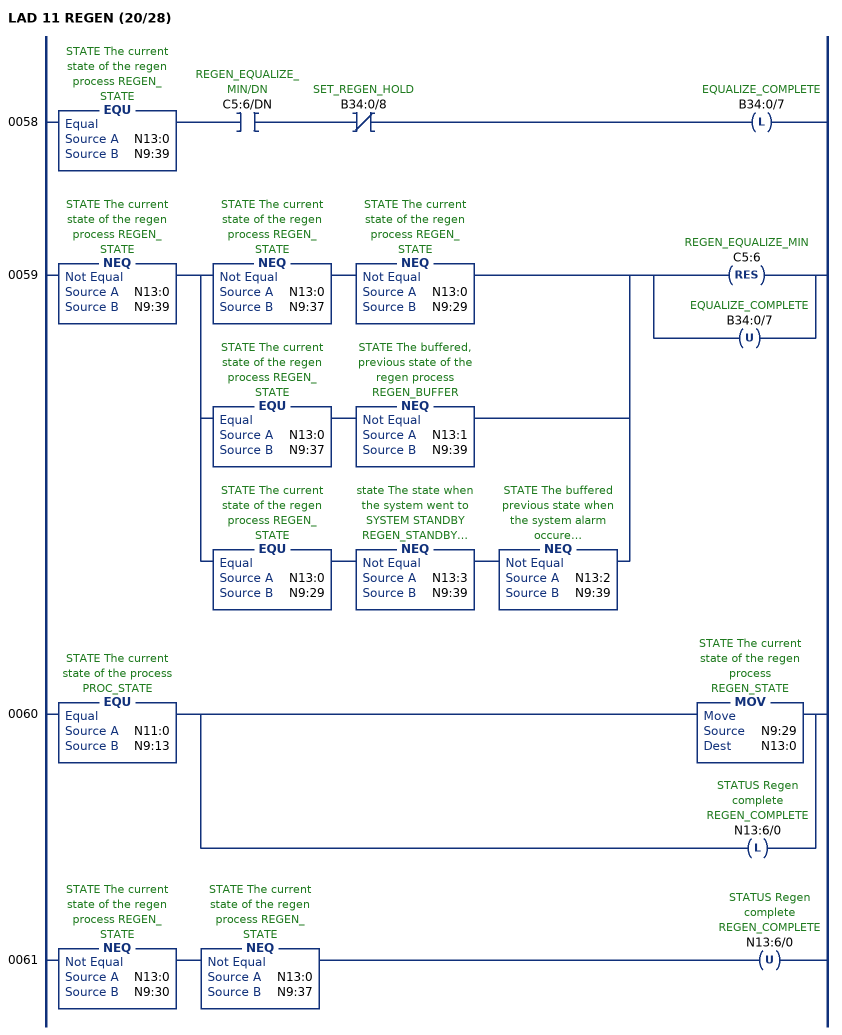
% Rung: 58 %
SOR EQU N13:0 N9:39 XIC C5:6/DN XIO B34:0/8 OTL B34:0/7 EOR
%   N13:0  REGEN_STATE  "STATE The current state of the regen process" %
%   N9:39  REGEN_EQUALIZE %
%   C5:6  REGEN_EQUALIZE_MIN %
%   B34:0/8  SET_REGEN_HOLD %
%   B34:0/7  EQUALIZE_COMPLETE %
% Rung: 59 %
SOR NEQ N13:0 N9:39 BST NEQ N13:0 N9:37 NEQ N13:0 N9:29 NXB EQU N13:0 N9:37 NEQ N13:1 N9:39 NXB EQU N13:0 N9:29 NEQ N13:3 N9:39 NEQ N13:2 N9:39 BND BST RES C5:6 NXB OTU B34:0/7 BND EOR
%   N13:0  REGEN_STATE  "STATE The current state of the regen process" %
%   N9:39  REGEN_EQUALIZE %
%   N9:37  REGEN_ALARM  "STATE Regen Alarm" %
%   N9:29  REGEN_IDLE %
%   N13:1  REGEN_BUFFER  "STATE The buffered, previous state of the regen process" %
%   N13:3  REGEN_STANDBY_BUFFER  "state The state when the system went to SYSTEM STANDBY" %
%   N13:2  REGEN_ALARM_BUFFER  "STATE The buffered previous state when the system alarm occured" %
%   C5:6  REGEN_EQUALIZE_MIN %
%   B34:0/7  EQUALIZE_COMPLETE %
% Rung: 60 %
SOR EQU N11:0 N9:13 BST MOV N9:29 N13:0 NXB OTL N13:6/0 BND EOR
%   N11:0  PROC_STATE  "STATE The current state of the process" %
%   N9:13  PROC_OVERLAP  "STATE Process Purify Overlap" %
%   N9:29  REGEN_IDLE %
%   N13:0  REGEN_STATE  "STATE The current state of the regen process" %
%   N13:6/0  REGEN_COMPLETE  "STATUS Regen complete" %
% Rung: 61 %
SOR NEQ N13:0 N9:30 NEQ N13:0 N9:37 OTU N13:6/0 EOR
%   N13:0  REGEN_STATE  "STATE The current state of the regen process" %
%   N9:30  REGEN_STANDBY  "STATE Regen Standby" %
%   N9:37  REGEN_ALARM  "STATE Regen Alarm" %
%   N13:6/0  REGEN_COMPLETE  "STATUS Regen complete" %

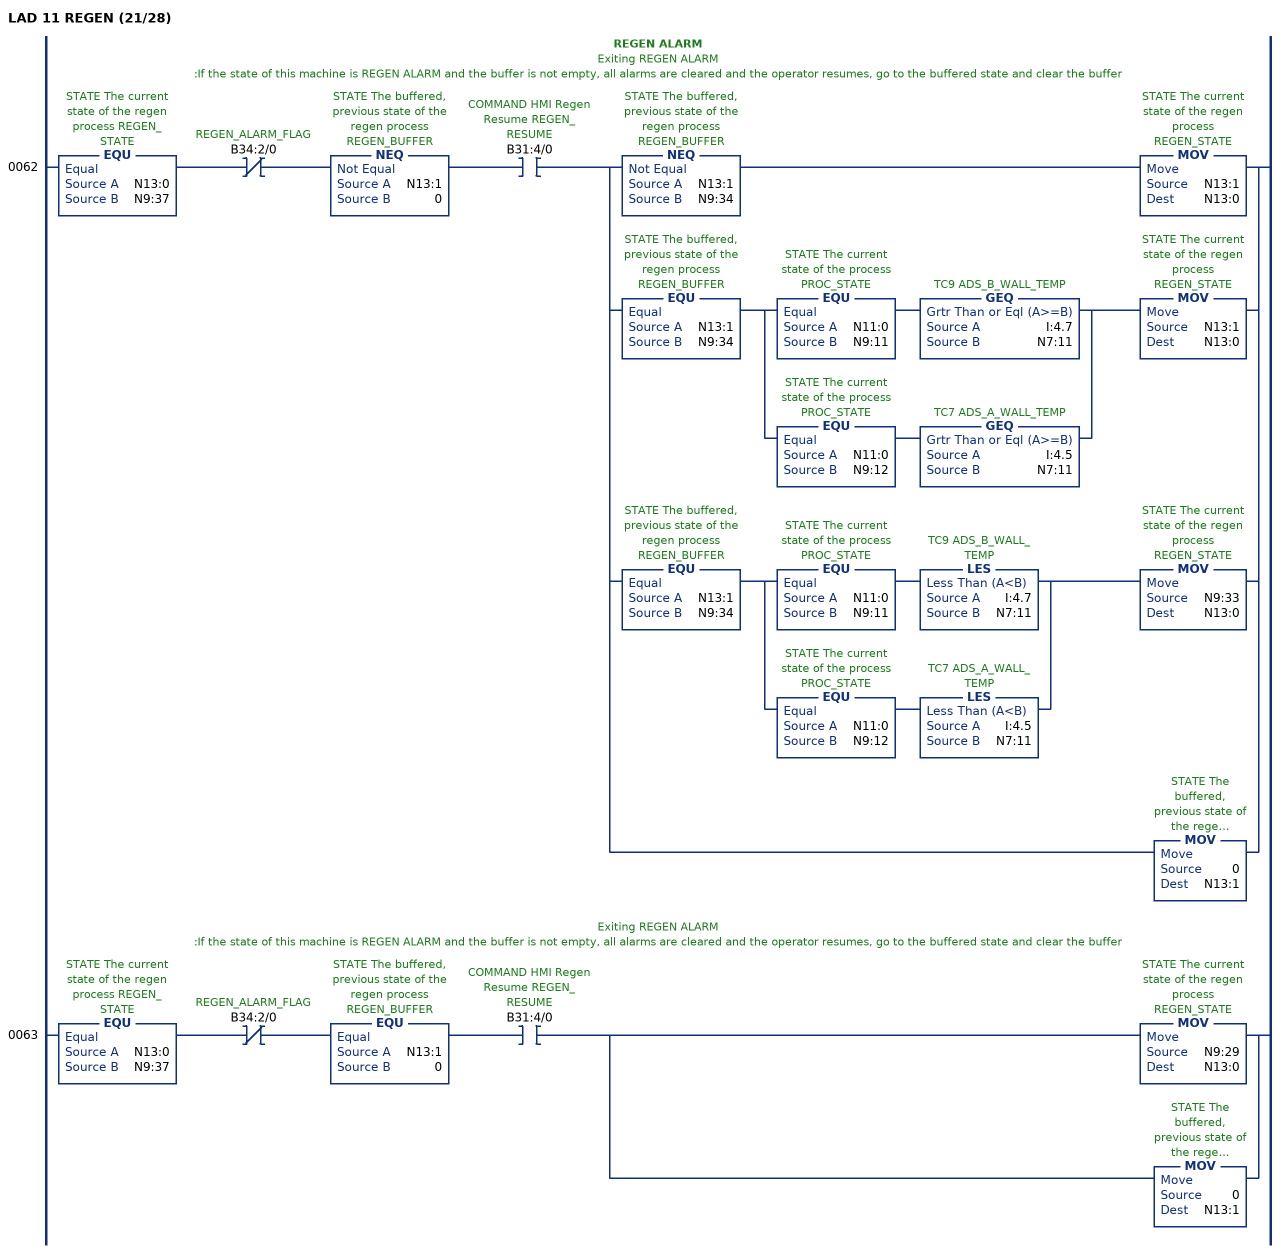
% Rung: 62 %
% TITLE: REGEN ALARM %
% Exiting REGEN ALARM
% :If the state of this machine is REGEN ALARM and the buffer is not empty, all alarms are cleared and the operator resumes, go to the buffered state and clear the buffer %
SOR EQU N13:0 N9:37 XIO B34:2/0 NEQ N13:1 0 XIC B31:4/0 BST NEQ N13:1 N9:34 MOV N13:1 N13:0 NXB EQU N13:1 N9:34 BST EQU N11:0 N9:11 GEQ I:4.7 N7:11 NXB EQU N11:0 N9:12 GEQ I:4.5 N7:11 BND MOV N13:1 N13:0 NXB EQU N13:1 N9:34 BST EQU N11:0 N9:11 LES I:4.7 N7:11 NXB EQU N11:0 N9:12 LES I:4.5 N7:11 BND MOV N9:33 N13:0 NXB MOV 0 N13:1 BND EOR
%   N13:0  REGEN_STATE  "STATE The current state of the regen process" %
%   N9:37  REGEN_ALARM  "STATE Regen Alarm" %
%   B34:2/0  REGEN_ALARM_FLAG %
%   N13:1  REGEN_BUFFER  "STATE The buffered, previous state of the regen process" %
%   B31:4/0  REGEN_RESUME  "COMMAND HMI Regen Resume" %
%   N9:34  REGEN_H2_REDUCTION  "STATE Regen Running" %
%   N11:0  PROC_STATE  "STATE The current state of the process" %
%   N9:11  PROC_PURIFY_A  "STATE Process Purify A" %
%   I:4.7  ADS_B_WALL_TEMP  "TC9" %
%   N7:11  ADS_BED_TEMP_HIGH  "CONFIG The temp at which the regen process may continue" %
%   N9:12  PROC_PURIFY_B  "STATE Process Purify B" %
%   I:4.5  ADS_A_WALL_TEMP  "TC7" %
%   N9:33  REGEN_HEAT_BED  "STATE Regen Heat wall" %
% Rung: 63 %
% Exiting REGEN ALARM
% :If the state of this machine is REGEN ALARM and the buffer is not empty, all alarms are cleared and the operator resumes, go to the buffered state and clear the buffer %
SOR EQU N13:0 N9:37 XIO B34:2/0 EQU N13:1 0 XIC B31:4/0 BST MOV N9:29 N13:0 NXB MOV 0 N13:1 BND EOR
%   N13:0  REGEN_STATE  "STATE The current state of the regen process" %
%   N9:37  REGEN_ALARM  "STATE Regen Alarm" %
%   B34:2/0  REGEN_ALARM_FLAG %
%   N13:1  REGEN_BUFFER  "STATE The buffered, previous state of the regen process" %
%   B31:4/0  REGEN_RESUME  "COMMAND HMI Regen Resume" %
%   N9:29  REGEN_IDLE %

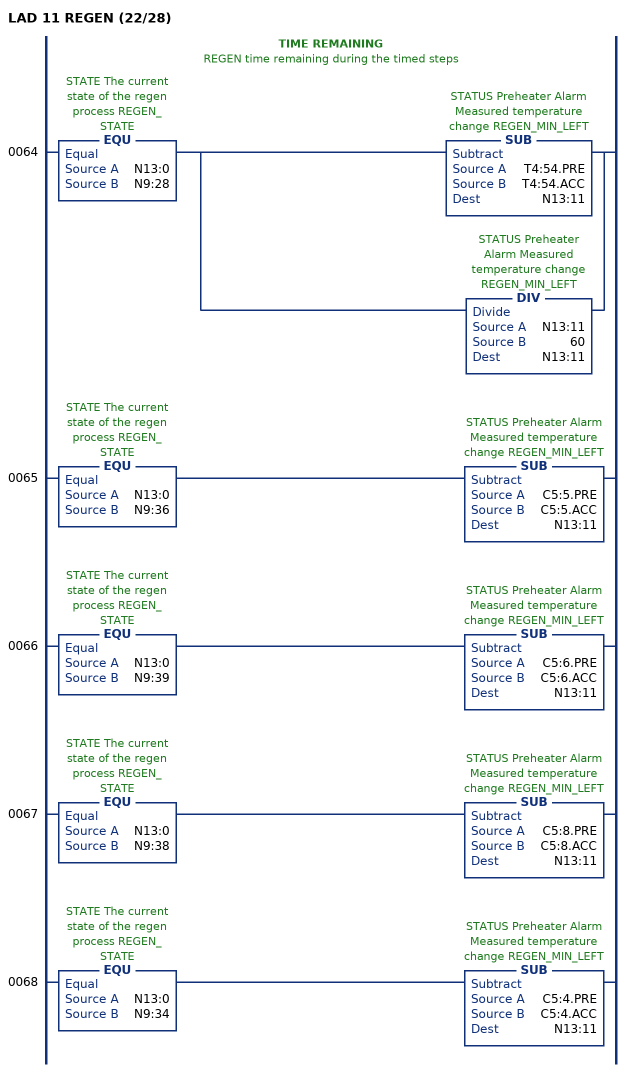
% Rung: 64 %
% TITLE: TIME REMAINING %
% REGEN time remaining during the timed steps %
SOR EQU N13:0 N9:28 BST SUB T4:54.PRE T4:54.ACC N13:11 NXB DIV N13:11 60 N13:11 BND EOR
%   N13:0  REGEN_STATE  "STATE The current state of the regen process" %
%   N9:28  REGEN_VENT_2  "STATE Regen Vent 2" %
%   T4:54  REGEN_VENT_2_TMR %
%   N13:11  REGEN_MIN_LEFT  "STATUS Preheater Alarm Measured temperature change" %
% Rung: 65 %
SOR EQU N13:0 N9:36 SUB C5:5.PRE C5:5.ACC N13:11 EOR
%   N13:0  REGEN_STATE  "STATE The current state of the regen process" %
%   N9:36  REGEN_COOL  "STATE Regen Cool" %
%   C5:5  REGEN_COOL_MINUTE  "COUNTER Regen the number of minutes for which the bed has cooled" %
%   N13:11  REGEN_MIN_LEFT  "STATUS Preheater Alarm Measured temperature change" %
% Rung: 66 %
SOR EQU N13:0 N9:39 SUB C5:6.PRE C5:6.ACC N13:11 EOR
%   N13:0  REGEN_STATE  "STATE The current state of the regen process" %
%   N9:39  REGEN_EQUALIZE %
%   C5:6  REGEN_EQUALIZE_MIN %
%   N13:11  REGEN_MIN_LEFT  "STATUS Preheater Alarm Measured temperature change" %
% Rung: 67 %
SOR EQU N13:0 N9:38 SUB C5:8.PRE C5:8.ACC N13:11 EOR
%   N13:0  REGEN_STATE  "STATE The current state of the regen process" %
%   N9:38  REGEN_PURGE  "STATE Regen Hot Purge" %
%   C5:8  REGEN_PURGE_MINUTES  "COUNTER Regen THe number of minutes the purge step runs" %
%   N13:11  REGEN_MIN_LEFT  "STATUS Preheater Alarm Measured temperature change" %
% Rung: 68 %
SOR EQU N13:0 N9:34 SUB C5:4.PRE C5:4.ACC N13:11 EOR
%   N13:0  REGEN_STATE  "STATE The current state of the regen process" %
%   N9:34  REGEN_H2_REDUCTION  "STATE Regen Running" %
%   C5:4  REGEN_REDUC_MINUTE  "COUNTER Regen The number of minutes which the regen reduc runs" %
%   N13:11  REGEN_MIN_LEFT  "STATUS Preheater Alarm Measured temperature change" %

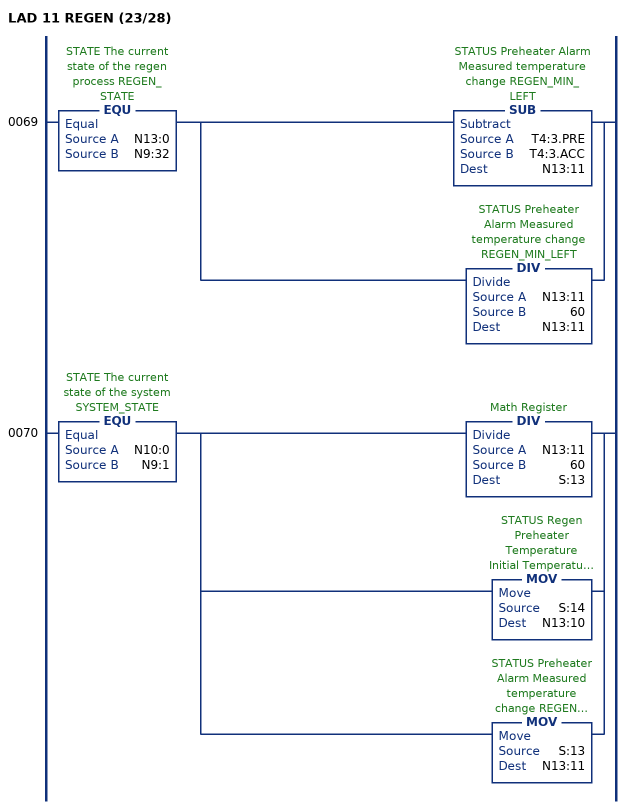
% Rung: 69 %
SOR EQU N13:0 N9:32 BST SUB T4:3.PRE T4:3.ACC N13:11 NXB DIV N13:11 60 N13:11 BND EOR
%   N13:0  REGEN_STATE  "STATE The current state of the regen process" %
%   N9:32  REGEN_VENT  "STATE Regen Vent" %
%   T4:3  REGEN_VENT_TIMER  "TIMER Regen Vent (seconds)" %
%   N13:11  REGEN_MIN_LEFT  "STATUS Preheater Alarm Measured temperature change" %
% Rung: 70 %
SOR EQU N10:0 N9:1 BST DIV N13:11 60 S:13 NXB MOV S:14 N13:10 NXB MOV S:13 N13:11 BND EOR
%   N10:0  SYSTEM_STATE  "STATE The current state of the system" %
%   N9:1  SYSTEM_PROCESS  "STATE System Process" %
%   N13:11  REGEN_MIN_LEFT  "STATUS Preheater Alarm Measured temperature change" %
%   S:13  "Math Register" %
%   S:14  "Math Register" %
%   N13:10  REGEN_HRS_LEFT  "STATUS Regen Preheater Temperature Initial Temperature" %

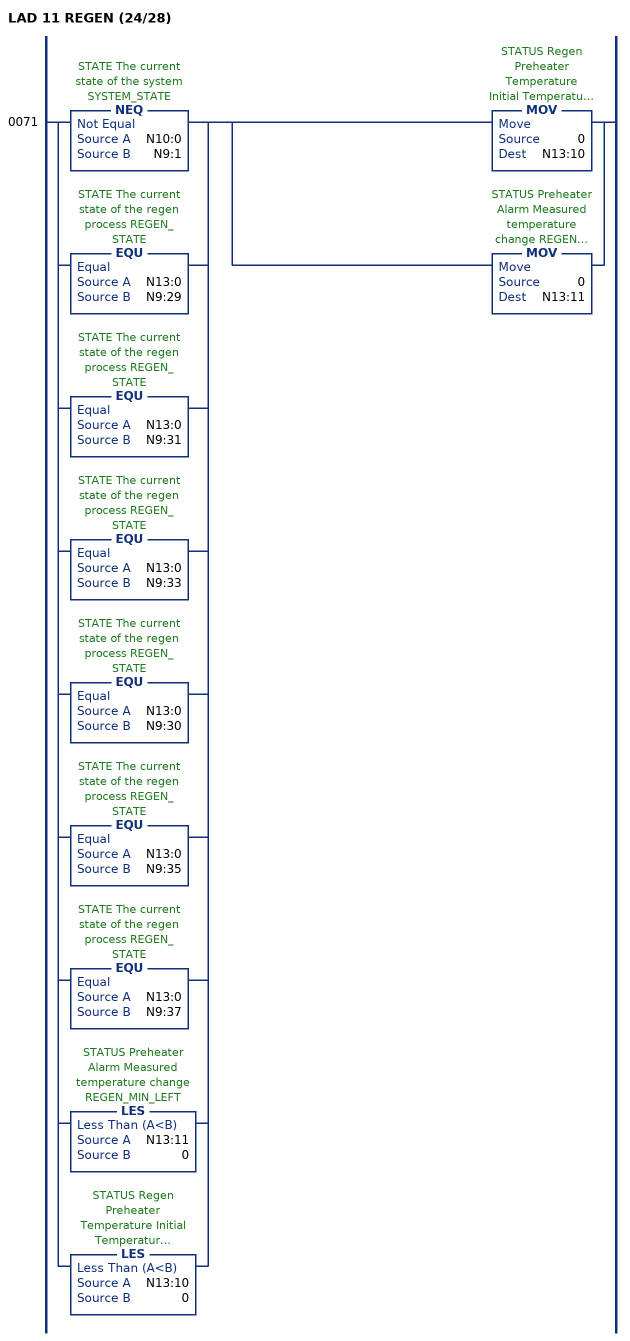
% Rung: 71 %
SOR BST NEQ N10:0 N9:1 NXB EQU N13:0 N9:29 NXB EQU N13:0 N9:31 NXB EQU N13:0 N9:33 NXB EQU N13:0 N9:30 NXB EQU N13:0 N9:35 NXB EQU N13:0 N9:37 NXB LES N13:11 0 NXB LES N13:10 0 BND BST MOV 0 N13:10 NXB MOV 0 N13:11 BND EOR
%   N10:0  SYSTEM_STATE  "STATE The current state of the system" %
%   N9:1  SYSTEM_PROCESS  "STATE System Process" %
%   N13:0  REGEN_STATE  "STATE The current state of the regen process" %
%   N9:29  REGEN_IDLE %
%   N9:31  REGEN_DELAY  "STATE Regen Delay" %
%   N9:33  REGEN_HEAT_BED  "STATE Regen Heat wall" %
%   N9:30  REGEN_STANDBY  "STATE Regen Standby" %
%   N9:35  REGEN_COOL_WALL  "STATE Regen Cool wall" %
%   N9:37  REGEN_ALARM  "STATE Regen Alarm" %
%   N13:11  REGEN_MIN_LEFT  "STATUS Preheater Alarm Measured temperature change" %
%   N13:10  REGEN_HRS_LEFT  "STATUS Regen Preheater Temperature Initial Temperature" %

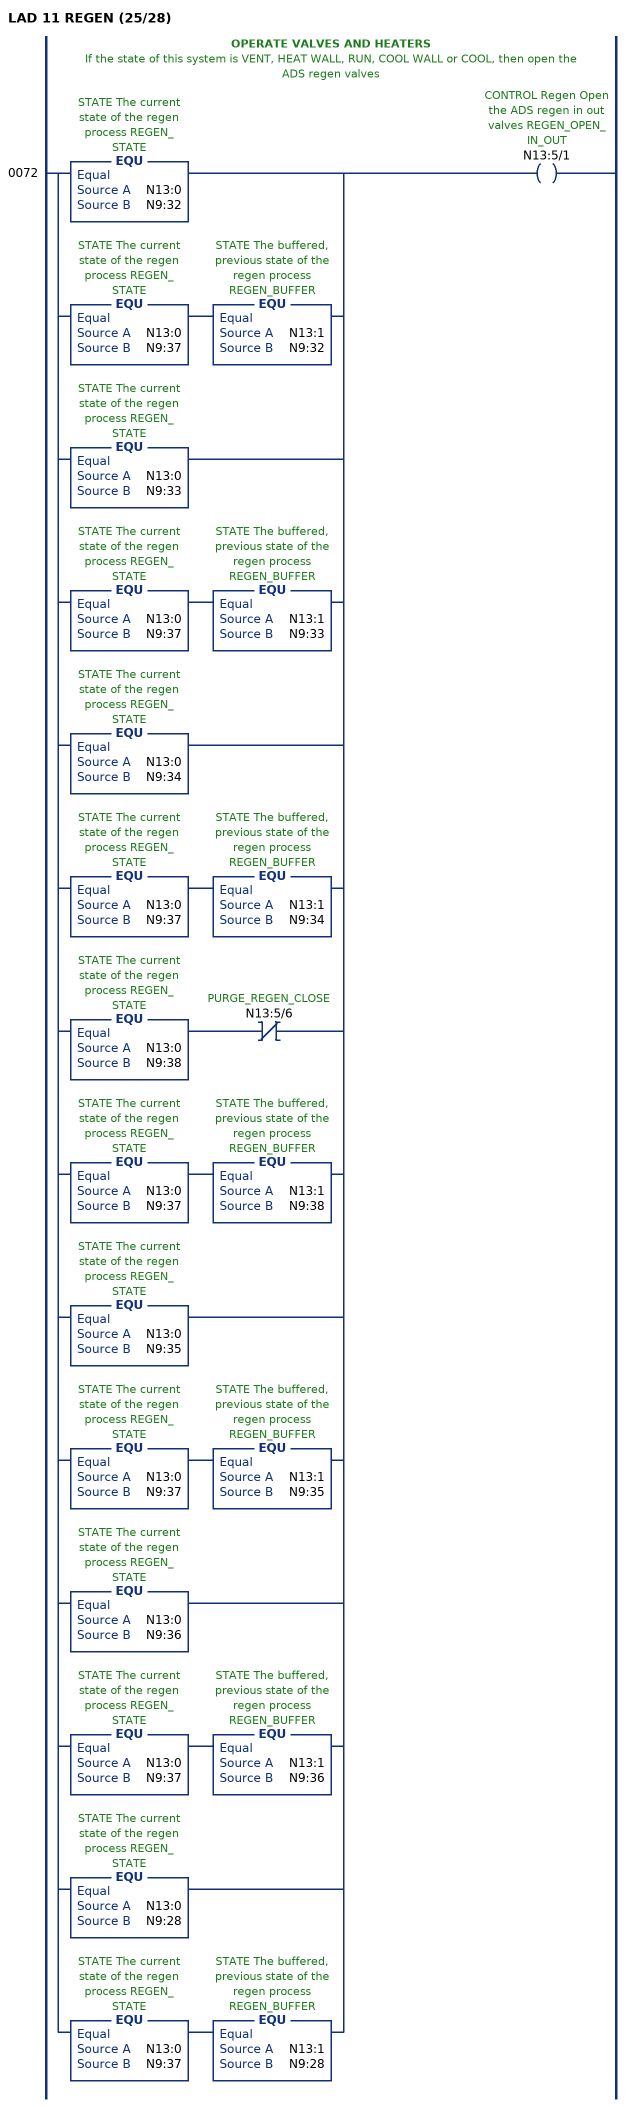
% Rung: 72 %
% TITLE: OPERATE VALVES AND HEATERS %
% If the state of this system is VENT, HEAT WALL, RUN, COOL WALL or COOL, then open the ADS regen valves %
SOR BST EQU N13:0 N9:32 NXB EQU N13:0 N9:37 EQU N13:1 N9:32 NXB EQU N13:0 N9:33 NXB EQU N13:0 N9:37 EQU N13:1 N9:33 NXB EQU N13:0 N9:34 NXB EQU N13:0 N9:37 EQU N13:1 N9:34 NXB EQU N13:0 N9:38 XIO N13:5/6 NXB EQU N13:0 N9:37 EQU N13:1 N9:38 NXB EQU N13:0 N9:35 NXB EQU N13:0 N9:37 EQU N13:1 N9:35 NXB EQU N13:0 N9:36 NXB EQU N13:0 N9:37 EQU N13:1 N9:36 NXB EQU N13:0 N9:28 NXB EQU N13:0 N9:37 EQU N13:1 N9:28 BND OTE N13:5/1 EOR
%   N13:0  REGEN_STATE  "STATE The current state of the regen process" %
%   N9:32  REGEN_VENT  "STATE Regen Vent" %
%   N9:37  REGEN_ALARM  "STATE Regen Alarm" %
%   N13:1  REGEN_BUFFER  "STATE The buffered, previous state of the regen process" %
%   N9:33  REGEN_HEAT_BED  "STATE Regen Heat wall" %
%   N9:34  REGEN_H2_REDUCTION  "STATE Regen Running" %
%   N9:38  REGEN_PURGE  "STATE Regen Hot Purge" %
%   N13:5/6  PURGE_REGEN_CLOSE %
%   N9:35  REGEN_COOL_WALL  "STATE Regen Cool wall" %
%   N9:36  REGEN_COOL  "STATE Regen Cool" %
%   N9:28  REGEN_VENT_2  "STATE Regen Vent 2" %
%   N13:5/1  REGEN_OPEN_IN_OUT  "CONTROL Regen Open the ADS regen in out valves" %

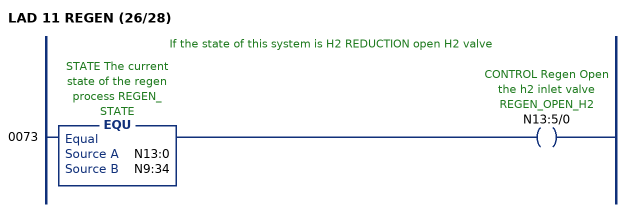
% Rung: 73 %
% If the state of this system is H2 REDUCTION open H2 valve %
SOR EQU N13:0 N9:34 OTE N13:5/0 EOR
%   N13:0  REGEN_STATE  "STATE The current state of the regen process" %
%   N9:34  REGEN_H2_REDUCTION  "STATE Regen Running" %
%   N13:5/0  REGEN_OPEN_H2  "CONTROL Regen Open the h2 inlet valve" %

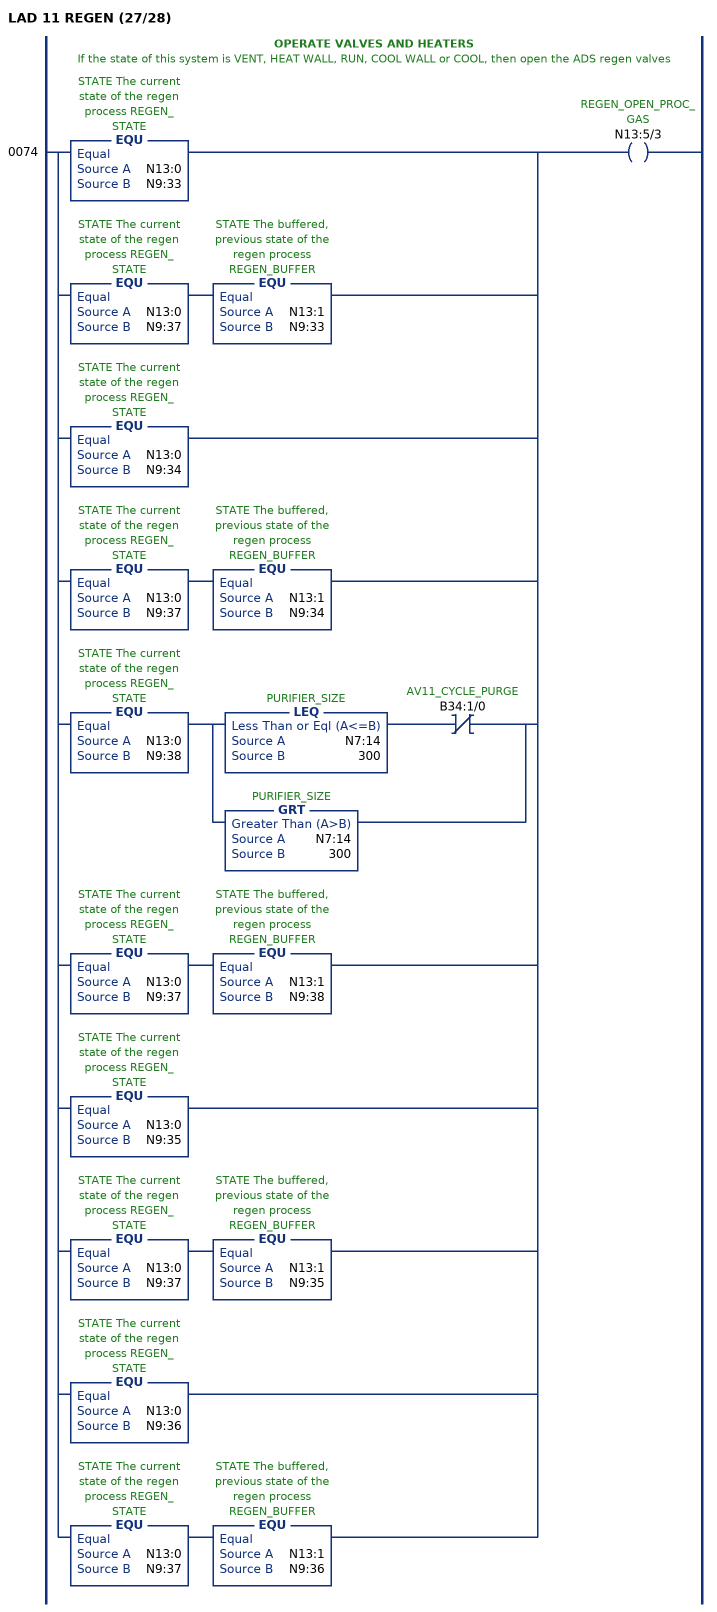
% Rung: 74 %
% TITLE: OPERATE VALVES AND HEATERS %
% If the state of this system is VENT, HEAT WALL, RUN, COOL WALL or COOL, then open the ADS regen valves %
SOR BST EQU N13:0 N9:33 NXB EQU N13:0 N9:37 EQU N13:1 N9:33 NXB EQU N13:0 N9:34 NXB EQU N13:0 N9:37 EQU N13:1 N9:34 NXB EQU N13:0 N9:38 BST LEQ N7:14 300 XIO B34:1/0 NXB GRT N7:14 300 BND NXB EQU N13:0 N9:37 EQU N13:1 N9:38 NXB EQU N13:0 N9:35 NXB EQU N13:0 N9:37 EQU N13:1 N9:35 NXB EQU N13:0 N9:36 NXB EQU N13:0 N9:37 EQU N13:1 N9:36 BND OTE N13:5/3 EOR
%   N13:0  REGEN_STATE  "STATE The current state of the regen process" %
%   N9:33  REGEN_HEAT_BED  "STATE Regen Heat wall" %
%   N9:37  REGEN_ALARM  "STATE Regen Alarm" %
%   N13:1  REGEN_BUFFER  "STATE The buffered, previous state of the regen process" %
%   N9:34  REGEN_H2_REDUCTION  "STATE Regen Running" %
%   N9:38  REGEN_PURGE  "STATE Regen Hot Purge" %
%   N7:14  PURIFIER_SIZE %
%   B34:1/0  AV11_CYCLE_PURGE %
%   N9:35  REGEN_COOL_WALL  "STATE Regen Cool wall" %
%   N9:36  REGEN_COOL  "STATE Regen Cool" %
%   N13:5/3  REGEN_OPEN_PROC_GAS %

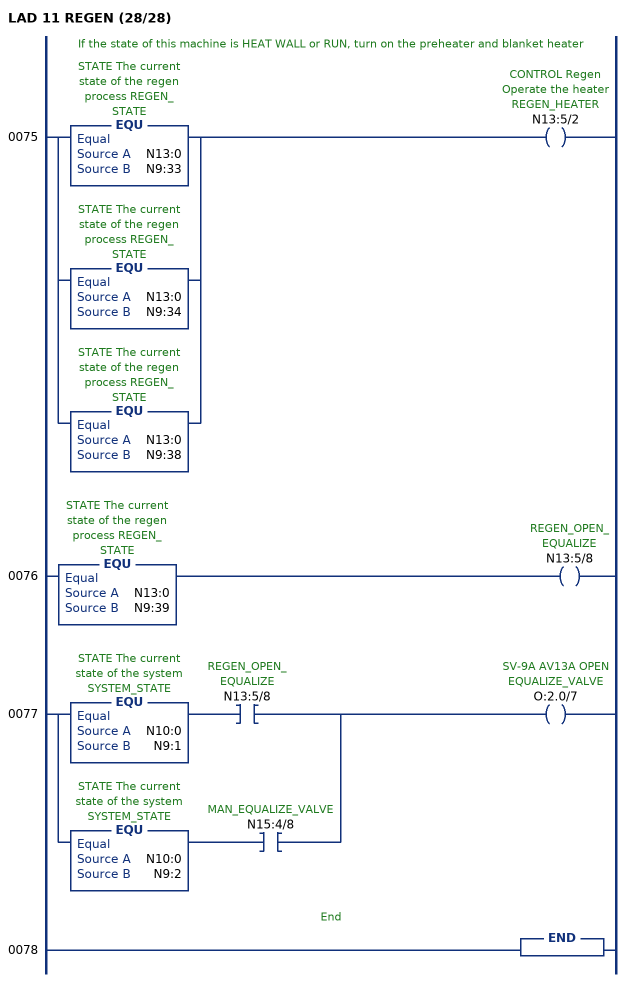
% Rung: 75 %
% If the state of this machine is HEAT WALL or RUN, turn on the preheater and blanket heater %
SOR BST EQU N13:0 N9:33 NXB EQU N13:0 N9:34 NXB EQU N13:0 N9:38 BND OTE N13:5/2 EOR
%   N13:0  REGEN_STATE  "STATE The current state of the regen process" %
%   N9:33  REGEN_HEAT_BED  "STATE Regen Heat wall" %
%   N9:34  REGEN_H2_REDUCTION  "STATE Regen Running" %
%   N9:38  REGEN_PURGE  "STATE Regen Hot Purge" %
%   N13:5/2  REGEN_HEATER  "CONTROL Regen Operate the heater" %
% Rung: 76 %
SOR EQU N13:0 N9:39 OTE N13:5/8 EOR
%   N13:0  REGEN_STATE  "STATE The current state of the regen process" %
%   N9:39  REGEN_EQUALIZE %
%   N13:5/8  REGEN_OPEN_EQUALIZE %
% Rung: 77 %
SOR BST EQU N10:0 N9:1 XIC N13:5/8 NXB EQU N10:0 N9:2 XIC N15:4/8 BND OTE O:2.0/7 EOR
%   N10:0  SYSTEM_STATE  "STATE The current state of the system" %
%   N9:1  SYSTEM_PROCESS  "STATE System Process" %
%   N13:5/8  REGEN_OPEN_EQUALIZE %
%   N9:2  SYSTEM_MANUAL  "STATE System Manual" %
%   N15:4/8  MAN_EQUALIZE_VALVE %
%   O:2.0/7  EQUALIZE_VALVE  "SV-9A AV13A OPEN" %
% Rung: 78 %
% End %
SOR END EOR

LADDER 12 "REGEN_FLT"    % regen alarms and warnings %
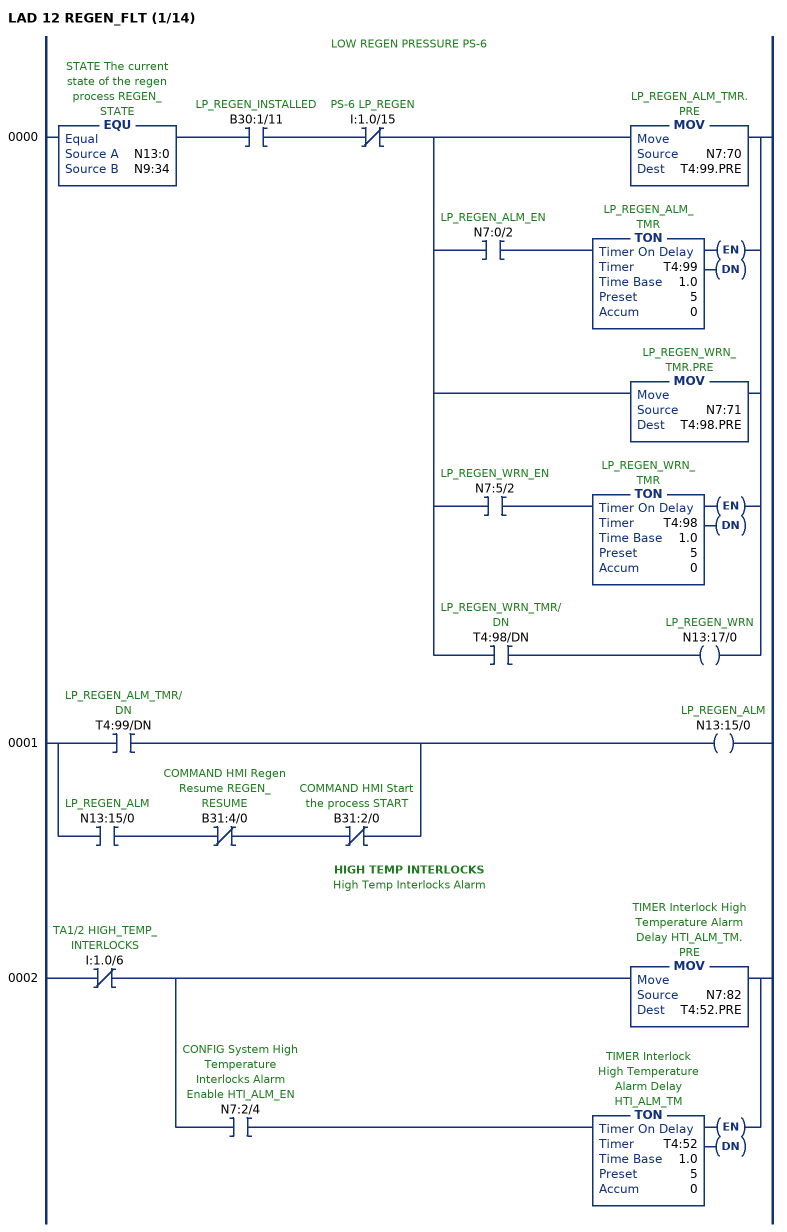
% Rung: 0 %
% LOW REGEN PRESSURE PS-6 %
SOR EQU N13:0 N9:34 XIC B30:1/11 XIO I:1.0/15 BST MOV N7:70 T4:99.PRE NXB XIC N7:0/2 TON T4:99 1.0 5 0 NXB MOV N7:71 T4:98.PRE NXB XIC N7:5/2 TON T4:98 1.0 5 0 NXB XIC T4:98/DN OTE N13:17/0 BND EOR
%   N13:0  REGEN_STATE  "STATE The current state of the regen process" %
%   N9:34  REGEN_H2_REDUCTION  "STATE Regen Running" %
%   B30:1/11  LP_REGEN_INSTALLED %
%   I:1.0/15  LP_REGEN  "PS-6" %
%   N7:70  LP_REGEN_ALM_DLY %
%   T4:99  LP_REGEN_ALM_TMR %
%   N7:0/2  LP_REGEN_ALM_EN %
%   N7:71  LP_REGEN_WRN_DLY %
%   T4:98  LP_REGEN_WRN_TMR %
%   N7:5/2  LP_REGEN_WRN_EN %
%   N13:17/0  LP_REGEN_WRN %
% Rung: 1 %
SOR BST XIC T4:99/DN NXB XIC N13:15/0 XIO B31:4/0 XIO B31:2/0 BND OTE N13:15/0 EOR
%   T4:99  LP_REGEN_ALM_TMR %
%   N13:15/0  LP_REGEN_ALM %
%   B31:4/0  REGEN_RESUME  "COMMAND HMI Regen Resume" %
%   B31:2/0  START  "COMMAND HMI Start the process" %
% Rung: 2 %
% TITLE: HIGH TEMP INTERLOCKS %
% High Temp Interlocks Alarm %
SOR XIO I:1.0/6 BST MOV N7:82 T4:52.PRE NXB XIC N7:2/4 TON T4:52 1.0 5 0 BND EOR
%   I:1.0/6  HIGH_TEMP_INTERLOCKS  "TA1/2" %
%   N7:82  HTI_ALM_DY  "CONFIG Interlocks High Temp Alarm Delay" %
%   T4:52  HTI_ALM_TM  "TIMER Interlock High Temperature Alarm Delay" %
%   N7:2/4  HTI_ALM_EN  "CONFIG System High Temperature Interlocks Alarm Enable" %

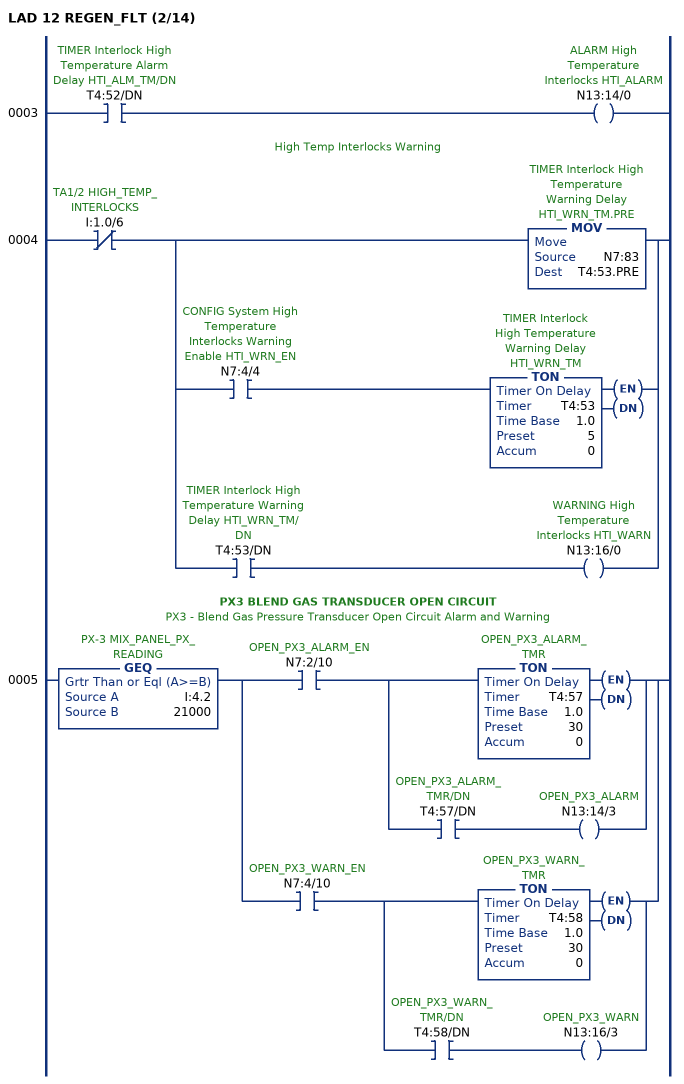
% Rung: 3 %
SOR XIC T4:52/DN OTE N13:14/0 EOR
%   T4:52  HTI_ALM_TM  "TIMER Interlock High Temperature Alarm Delay" %
%   N13:14/0  HTI_ALARM  "ALARM High Temperature Interlocks" %
% Rung: 4 %
% High Temp Interlocks Warning %
SOR XIO I:1.0/6 BST MOV N7:83 T4:53.PRE NXB XIC N7:4/4 TON T4:53 1.0 5 0 NXB XIC T4:53/DN OTE N13:16/0 BND EOR
%   I:1.0/6  HIGH_TEMP_INTERLOCKS  "TA1/2" %
%   N7:83  HTI_WRN_DY  "CONFIG Interlocks High Temp Warning Delay" %
%   T4:53  HTI_WRN_TM  "TIMER Interlock High Temperature Warning Delay" %
%   N7:4/4  HTI_WRN_EN  "CONFIG System High Temperature Interlocks Warning Enable" %
%   N13:16/0  HTI_WARN  "WARNING High Temperature Interlocks" %
% Rung: 5 %
% TITLE: PX3 BLEND GAS TRANSDUCER OPEN CIRCUIT %
% PX3 - Blend Gas Pressure Transducer Open Circuit Alarm and Warning %
SOR GEQ I:4.2 21000 BST XIC N7:2/10 BST TON T4:57 1.0 30 0 NXB XIC T4:57/DN OTE N13:14/3 BND NXB XIC N7:4/10 BST TON T4:58 1.0 30 0 NXB XIC T4:58/DN OTE N13:16/3 BND BND EOR
%   I:4.2  MIX_PANEL_PX_READING  "PX-3" %
%   N7:2/10  OPEN_PX3_ALARM_EN %
%   T4:57  OPEN_PX3_ALARM_TMR %
%   N13:14/3  OPEN_PX3_ALARM %
%   N7:4/10  OPEN_PX3_WARN_EN %
%   T4:58  OPEN_PX3_WARN_TMR %
%   N13:16/3  OPEN_PX3_WARN %

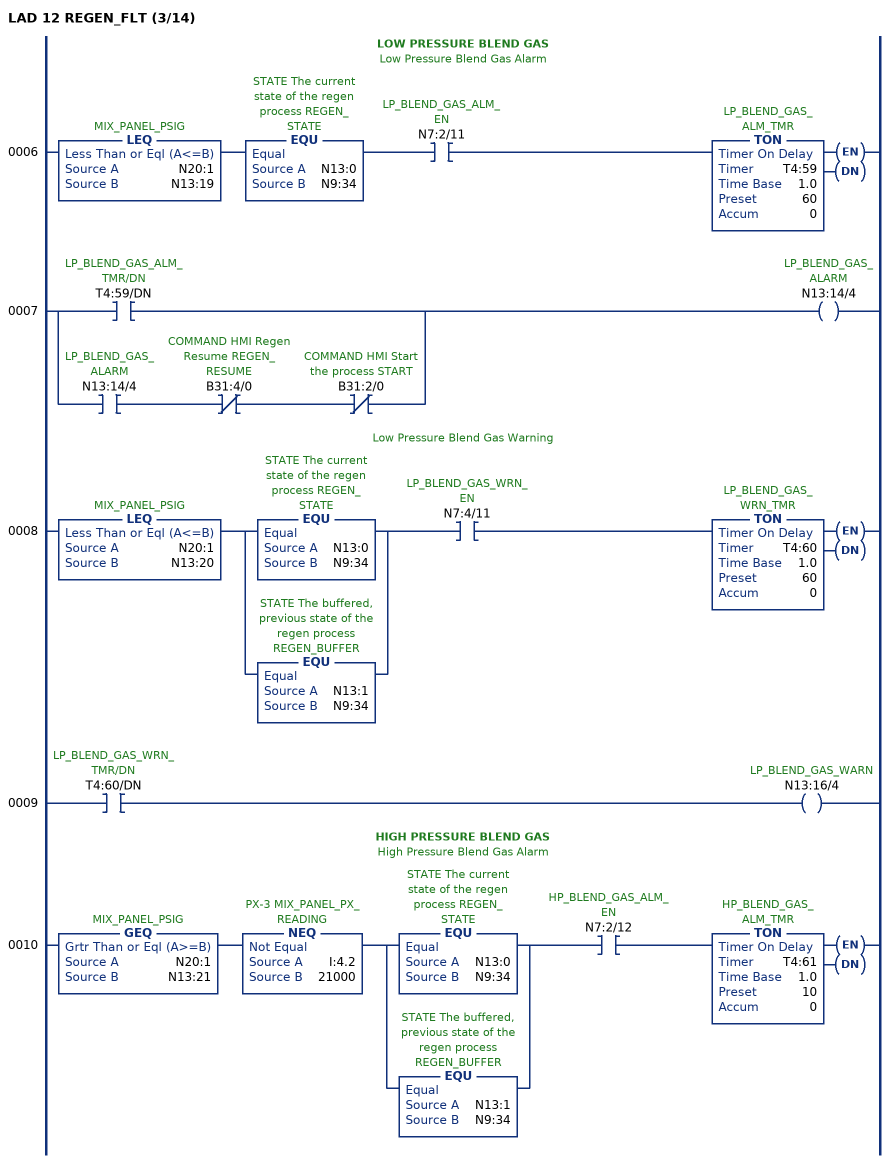
% Rung: 6 %
% TITLE: LOW PRESSURE BLEND GAS %
% Low Pressure Blend Gas Alarm %
SOR LEQ N20:1 N13:19 EQU N13:0 N9:34 XIC N7:2/11 TON T4:59 1.0 60 0 EOR
%   N20:1  MIX_PANEL_PSIG %
%   N13:19  LP_BLEND_GAS_ALM_SP %
%   N13:0  REGEN_STATE  "STATE The current state of the regen process" %
%   N9:34  REGEN_H2_REDUCTION  "STATE Regen Running" %
%   N7:2/11  LP_BLEND_GAS_ALM_EN %
%   T4:59  LP_BLEND_GAS_ALM_TMR %
% Rung: 7 %
SOR BST XIC T4:59/DN NXB XIC N13:14/4 XIO B31:4/0 XIO B31:2/0 BND OTE N13:14/4 EOR
%   T4:59  LP_BLEND_GAS_ALM_TMR %
%   N13:14/4  LP_BLEND_GAS_ALARM %
%   B31:4/0  REGEN_RESUME  "COMMAND HMI Regen Resume" %
%   B31:2/0  START  "COMMAND HMI Start the process" %
% Rung: 8 %
% Low Pressure Blend Gas Warning %
SOR LEQ N20:1 N13:20 BST EQU N13:0 N9:34 NXB EQU N13:1 N9:34 BND XIC N7:4/11 TON T4:60 1.0 60 0 EOR
%   N20:1  MIX_PANEL_PSIG %
%   N13:20  LP_BLEND_GAS_WRN_SP %
%   N13:0  REGEN_STATE  "STATE The current state of the regen process" %
%   N9:34  REGEN_H2_REDUCTION  "STATE Regen Running" %
%   N13:1  REGEN_BUFFER  "STATE The buffered, previous state of the regen process" %
%   N7:4/11  LP_BLEND_GAS_WRN_EN %
%   T4:60  LP_BLEND_GAS_WRN_TMR %
% Rung: 9 %
SOR XIC T4:60/DN OTE N13:16/4 EOR
%   T4:60  LP_BLEND_GAS_WRN_TMR %
%   N13:16/4  LP_BLEND_GAS_WARN %
% Rung: 10 %
% TITLE: HIGH PRESSURE BLEND GAS %
% High Pressure Blend Gas Alarm %
SOR GEQ N20:1 N13:21 NEQ I:4.2 21000 BST EQU N13:0 N9:34 NXB EQU N13:1 N9:34 BND XIC N7:2/12 TON T4:61 1.0 10 0 EOR
%   N20:1  MIX_PANEL_PSIG %
%   N13:21  HP_BLEND_GAS_ALM_SP %
%   I:4.2  MIX_PANEL_PX_READING  "PX-3" %
%   N13:0  REGEN_STATE  "STATE The current state of the regen process" %
%   N9:34  REGEN_H2_REDUCTION  "STATE Regen Running" %
%   N13:1  REGEN_BUFFER  "STATE The buffered, previous state of the regen process" %
%   N7:2/12  HP_BLEND_GAS_ALM_EN %
%   T4:61  HP_BLEND_GAS_ALM_TMR %

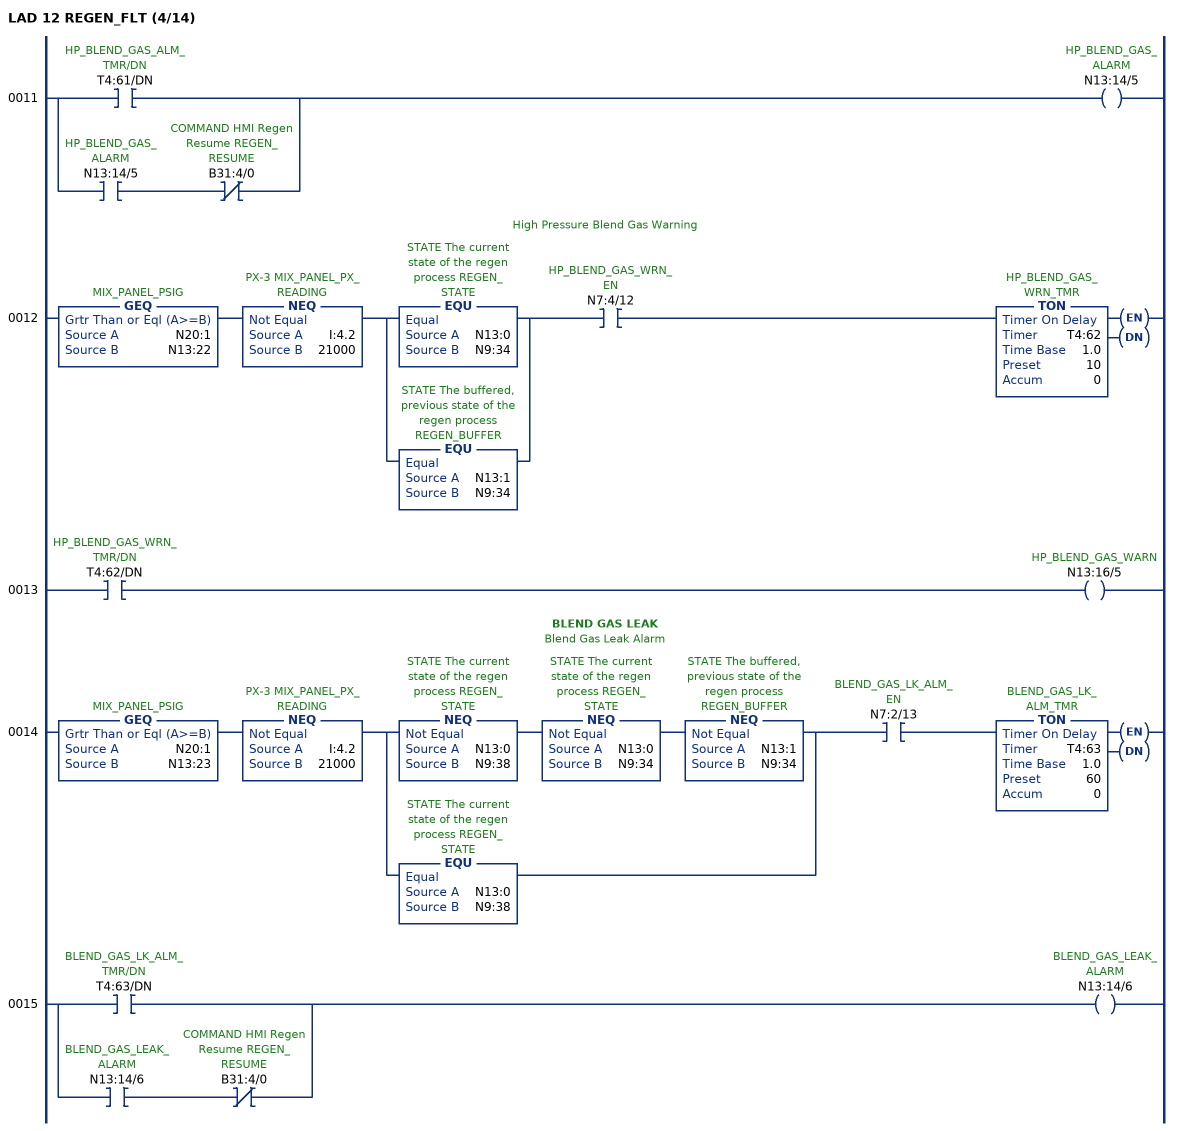
% Rung: 11 %
SOR BST XIC T4:61/DN NXB XIC N13:14/5 XIO B31:4/0 BND OTE N13:14/5 EOR
%   T4:61  HP_BLEND_GAS_ALM_TMR %
%   N13:14/5  HP_BLEND_GAS_ALARM %
%   B31:4/0  REGEN_RESUME  "COMMAND HMI Regen Resume" %
% Rung: 12 %
% High Pressure Blend Gas Warning %
SOR GEQ N20:1 N13:22 NEQ I:4.2 21000 BST EQU N13:0 N9:34 NXB EQU N13:1 N9:34 BND XIC N7:4/12 TON T4:62 1.0 10 0 EOR
%   N20:1  MIX_PANEL_PSIG %
%   N13:22  HP_BLEND_GAS_WRN_SP %
%   I:4.2  MIX_PANEL_PX_READING  "PX-3" %
%   N13:0  REGEN_STATE  "STATE The current state of the regen process" %
%   N9:34  REGEN_H2_REDUCTION  "STATE Regen Running" %
%   N13:1  REGEN_BUFFER  "STATE The buffered, previous state of the regen process" %
%   N7:4/12  HP_BLEND_GAS_WRN_EN %
%   T4:62  HP_BLEND_GAS_WRN_TMR %
% Rung: 13 %
SOR XIC T4:62/DN OTE N13:16/5 EOR
%   T4:62  HP_BLEND_GAS_WRN_TMR %
%   N13:16/5  HP_BLEND_GAS_WARN %
% Rung: 14 %
% TITLE: BLEND GAS LEAK %
% Blend Gas Leak Alarm %
SOR GEQ N20:1 N13:23 NEQ I:4.2 21000 BST NEQ N13:0 N9:38 NEQ N13:0 N9:34 NEQ N13:1 N9:34 NXB EQU N13:0 N9:38 BND XIC N7:2/13 TON T4:63 1.0 60 0 EOR
%   N20:1  MIX_PANEL_PSIG %
%   N13:23  BLEND_GAS_LK_ALM_SP %
%   I:4.2  MIX_PANEL_PX_READING  "PX-3" %
%   N13:0  REGEN_STATE  "STATE The current state of the regen process" %
%   N9:38  REGEN_PURGE  "STATE Regen Hot Purge" %
%   N9:34  REGEN_H2_REDUCTION  "STATE Regen Running" %
%   N13:1  REGEN_BUFFER  "STATE The buffered, previous state of the regen process" %
%   N7:2/13  BLEND_GAS_LK_ALM_EN %
%   T4:63  BLEND_GAS_LK_ALM_TMR %
% Rung: 15 %
SOR BST XIC T4:63/DN NXB XIC N13:14/6 XIO B31:4/0 BND OTE N13:14/6 EOR
%   T4:63  BLEND_GAS_LK_ALM_TMR %
%   N13:14/6  BLEND_GAS_LEAK_ALARM %
%   B31:4/0  REGEN_RESUME  "COMMAND HMI Regen Resume" %

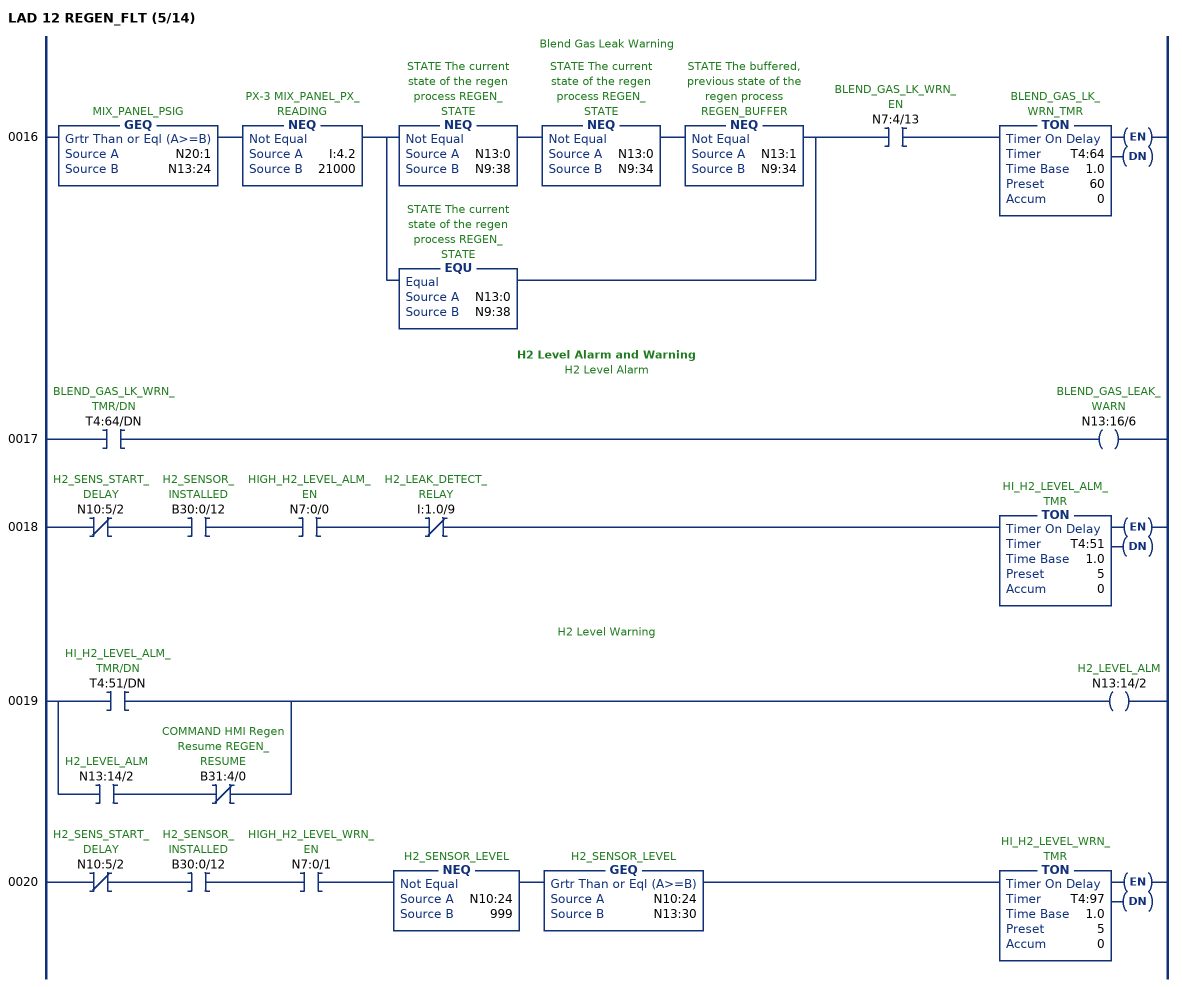
% Rung: 16 %
% Blend Gas Leak Warning %
SOR GEQ N20:1 N13:24 NEQ I:4.2 21000 BST NEQ N13:0 N9:38 NEQ N13:0 N9:34 NEQ N13:1 N9:34 NXB EQU N13:0 N9:38 BND XIC N7:4/13 TON T4:64 1.0 60 0 EOR
%   N20:1  MIX_PANEL_PSIG %
%   N13:24  BLEND_GAS_LK_WRN_SP %
%   I:4.2  MIX_PANEL_PX_READING  "PX-3" %
%   N13:0  REGEN_STATE  "STATE The current state of the regen process" %
%   N9:38  REGEN_PURGE  "STATE Regen Hot Purge" %
%   N9:34  REGEN_H2_REDUCTION  "STATE Regen Running" %
%   N13:1  REGEN_BUFFER  "STATE The buffered, previous state of the regen process" %
%   N7:4/13  BLEND_GAS_LK_WRN_EN %
%   T4:64  BLEND_GAS_LK_WRN_TMR %
% Rung: 17 %
% TITLE: H2 Level Alarm and Warning %
% H2 Level Alarm %
SOR XIC T4:64/DN OTE N13:16/6 EOR
%   T4:64  BLEND_GAS_LK_WRN_TMR %
%   N13:16/6  BLEND_GAS_LEAK_WARN %
% Rung: 18 %
SOR XIO N10:5/2 XIC B30:0/12 XIC N7:0/0 XIO I:1.0/9 TON T4:51 1.0 5 0 EOR
%   N10:5/2  H2_SENS_START_DELAY %
%   B30:0/12  H2_SENSOR_INSTALLED %
%   N7:0/0  HIGH_H2_LEVEL_ALM_EN %
%   I:1.0/9  H2_LEAK_DETECT_RELAY %
%   T4:51  HI_H2_LEVEL_ALM_TMR %
% Rung: 19 %
% H2 Level Warning %
SOR BST XIC T4:51/DN NXB XIC N13:14/2 XIO B31:4/0 BND OTE N13:14/2 EOR
%   T4:51  HI_H2_LEVEL_ALM_TMR %
%   N13:14/2  H2_LEVEL_ALM %
%   B31:4/0  REGEN_RESUME  "COMMAND HMI Regen Resume" %
% Rung: 20 %
SOR XIO N10:5/2 XIC B30:0/12 XIC N7:0/1 NEQ N10:24 999 GEQ N10:24 N13:30 TON T4:97 1.0 5 0 EOR
%   N10:5/2  H2_SENS_START_DELAY %
%   B30:0/12  H2_SENSOR_INSTALLED %
%   N7:0/1  HIGH_H2_LEVEL_WRN_EN %
%   N10:24  H2_SENSOR_LEVEL %
%   N13:30  HIGH_H2_LEVEL_WRN_SP %
%   T4:97  HI_H2_LEVEL_WRN_TMR %

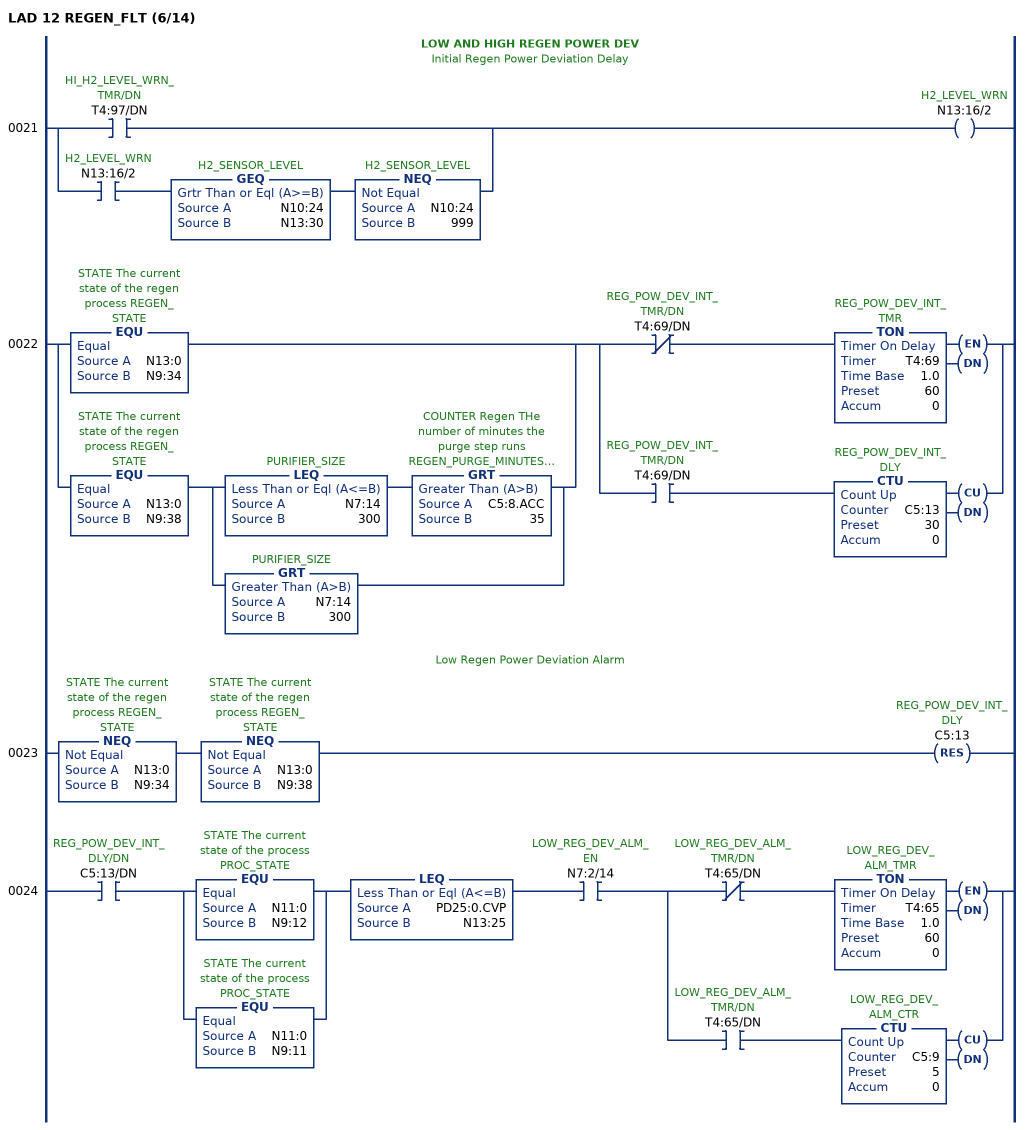
% Rung: 21 %
% TITLE: LOW AND HIGH REGEN POWER DEV %
% Initial Regen Power Deviation Delay %
SOR BST XIC T4:97/DN NXB XIC N13:16/2 GEQ N10:24 N13:30 NEQ N10:24 999 BND OTE N13:16/2 EOR
%   T4:97  HI_H2_LEVEL_WRN_TMR %
%   N13:16/2  H2_LEVEL_WRN %
%   N10:24  H2_SENSOR_LEVEL %
%   N13:30  HIGH_H2_LEVEL_WRN_SP %
% Rung: 22 %
SOR BST EQU N13:0 N9:34 NXB EQU N13:0 N9:38 BST LEQ N7:14 300 GRT C5:8.ACC 35 NXB GRT N7:14 300 BND BND BST XIO T4:69/DN TON T4:69 1.0 60 0 NXB XIC T4:69/DN CTU C5:13 30 0 BND EOR
%   N13:0  REGEN_STATE  "STATE The current state of the regen process" %
%   N9:34  REGEN_H2_REDUCTION  "STATE Regen Running" %
%   N9:38  REGEN_PURGE  "STATE Regen Hot Purge" %
%   N7:14  PURIFIER_SIZE %
%   C5:8  REGEN_PURGE_MINUTES  "COUNTER Regen THe number of minutes the purge step runs" %
%   T4:69  REG_POW_DEV_INT_TMR %
%   C5:13  REG_POW_DEV_INT_DLY %
% Rung: 23 %
% Low Regen Power Deviation Alarm %
SOR NEQ N13:0 N9:34 NEQ N13:0 N9:38 RES C5:13 EOR
%   N13:0  REGEN_STATE  "STATE The current state of the regen process" %
%   N9:34  REGEN_H2_REDUCTION  "STATE Regen Running" %
%   N9:38  REGEN_PURGE  "STATE Regen Hot Purge" %
%   C5:13  REG_POW_DEV_INT_DLY %
% Rung: 24 %
SOR XIC C5:13/DN BST EQU N11:0 N9:12 NXB EQU N11:0 N9:11 BND LEQ PD25:0.CVP N13:25 XIC N7:2/14 BST XIO T4:65/DN TON T4:65 1.0 60 0 NXB XIC T4:65/DN CTU C5:9 5 0 BND EOR
%   C5:13  REG_POW_DEV_INT_DLY %
%   N11:0  PROC_STATE  "STATE The current state of the process" %
%   N9:12  PROC_PURIFY_B  "STATE Process Purify B" %
%   N9:11  PROC_PURIFY_A  "STATE Process Purify A" %
%   N13:25  LOW_REG_DEV_ALM_SP %
%   N7:2/14  LOW_REG_DEV_ALM_EN %
%   T4:65  LOW_REG_DEV_ALM_TMR %
%   C5:9  LOW_REG_DEV_ALM_CTR %

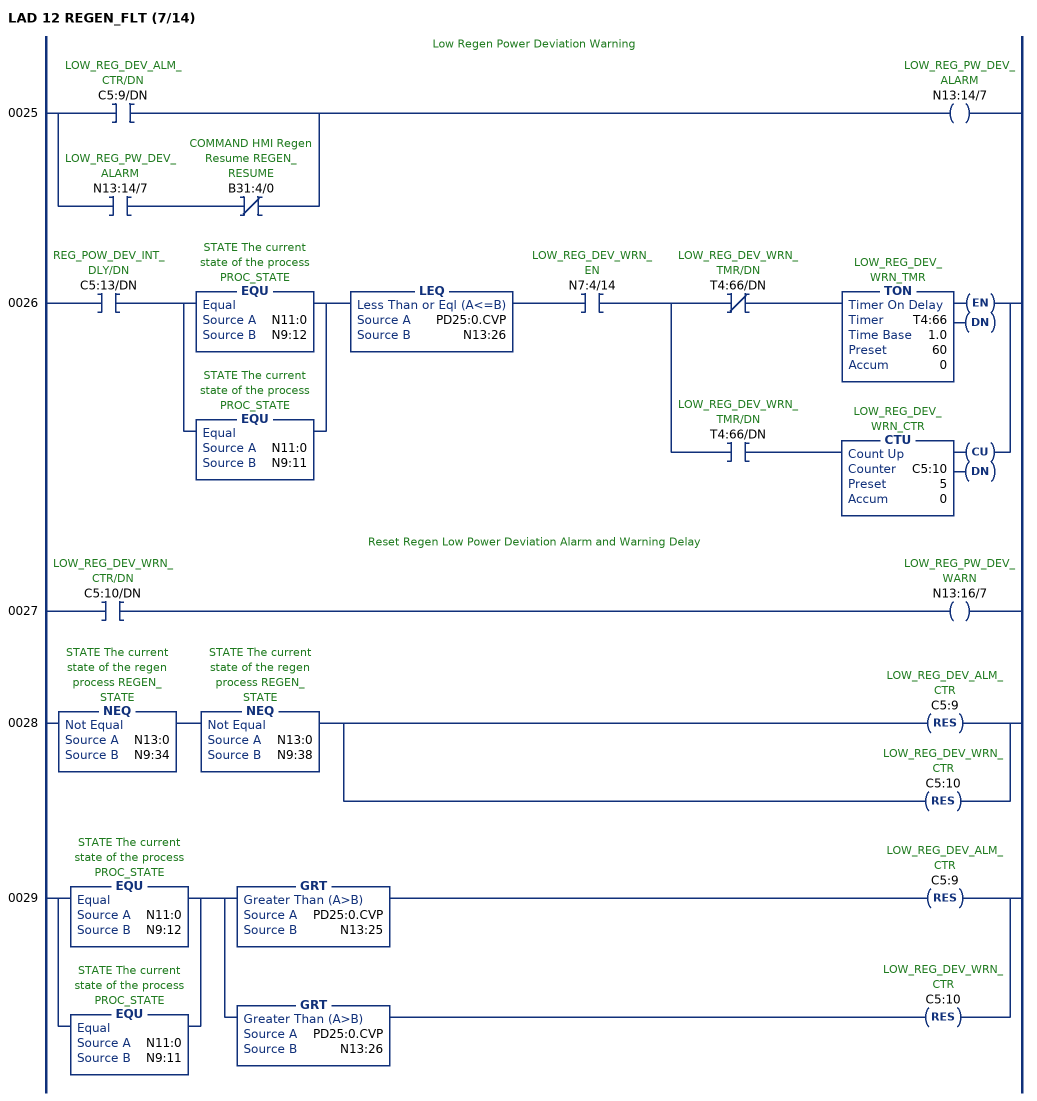
% Rung: 25 %
% Low Regen Power Deviation Warning %
SOR BST XIC C5:9/DN NXB XIC N13:14/7 XIO B31:4/0 BND OTE N13:14/7 EOR
%   C5:9  LOW_REG_DEV_ALM_CTR %
%   N13:14/7  LOW_REG_PW_DEV_ALARM %
%   B31:4/0  REGEN_RESUME  "COMMAND HMI Regen Resume" %
% Rung: 26 %
SOR XIC C5:13/DN BST EQU N11:0 N9:12 NXB EQU N11:0 N9:11 BND LEQ PD25:0.CVP N13:26 XIC N7:4/14 BST XIO T4:66/DN TON T4:66 1.0 60 0 NXB XIC T4:66/DN CTU C5:10 5 0 BND EOR
%   C5:13  REG_POW_DEV_INT_DLY %
%   N11:0  PROC_STATE  "STATE The current state of the process" %
%   N9:12  PROC_PURIFY_B  "STATE Process Purify B" %
%   N9:11  PROC_PURIFY_A  "STATE Process Purify A" %
%   N13:26  LOW_REG_DEV_WRN_SP %
%   N7:4/14  LOW_REG_DEV_WRN_EN %
%   T4:66  LOW_REG_DEV_WRN_TMR %
%   C5:10  LOW_REG_DEV_WRN_CTR %
% Rung: 27 %
% Reset Regen Low Power Deviation Alarm and Warning Delay %
SOR XIC C5:10/DN OTE N13:16/7 EOR
%   C5:10  LOW_REG_DEV_WRN_CTR %
%   N13:16/7  LOW_REG_PW_DEV_WARN %
% Rung: 28 %
SOR NEQ N13:0 N9:34 NEQ N13:0 N9:38 BST RES C5:9 NXB RES C5:10 BND EOR
%   N13:0  REGEN_STATE  "STATE The current state of the regen process" %
%   N9:34  REGEN_H2_REDUCTION  "STATE Regen Running" %
%   N9:38  REGEN_PURGE  "STATE Regen Hot Purge" %
%   C5:9  LOW_REG_DEV_ALM_CTR %
%   C5:10  LOW_REG_DEV_WRN_CTR %
% Rung: 29 %
SOR BST EQU N11:0 N9:12 NXB EQU N11:0 N9:11 BND BST GRT PD25:0.CVP N13:25 RES C5:9 NXB GRT PD25:0.CVP N13:26 RES C5:10 BND EOR
%   N11:0  PROC_STATE  "STATE The current state of the process" %
%   N9:12  PROC_PURIFY_B  "STATE Process Purify B" %
%   N9:11  PROC_PURIFY_A  "STATE Process Purify A" %
%   N13:25  LOW_REG_DEV_ALM_SP %
%   C5:9  LOW_REG_DEV_ALM_CTR %
%   N13:26  LOW_REG_DEV_WRN_SP %
%   C5:10  LOW_REG_DEV_WRN_CTR %

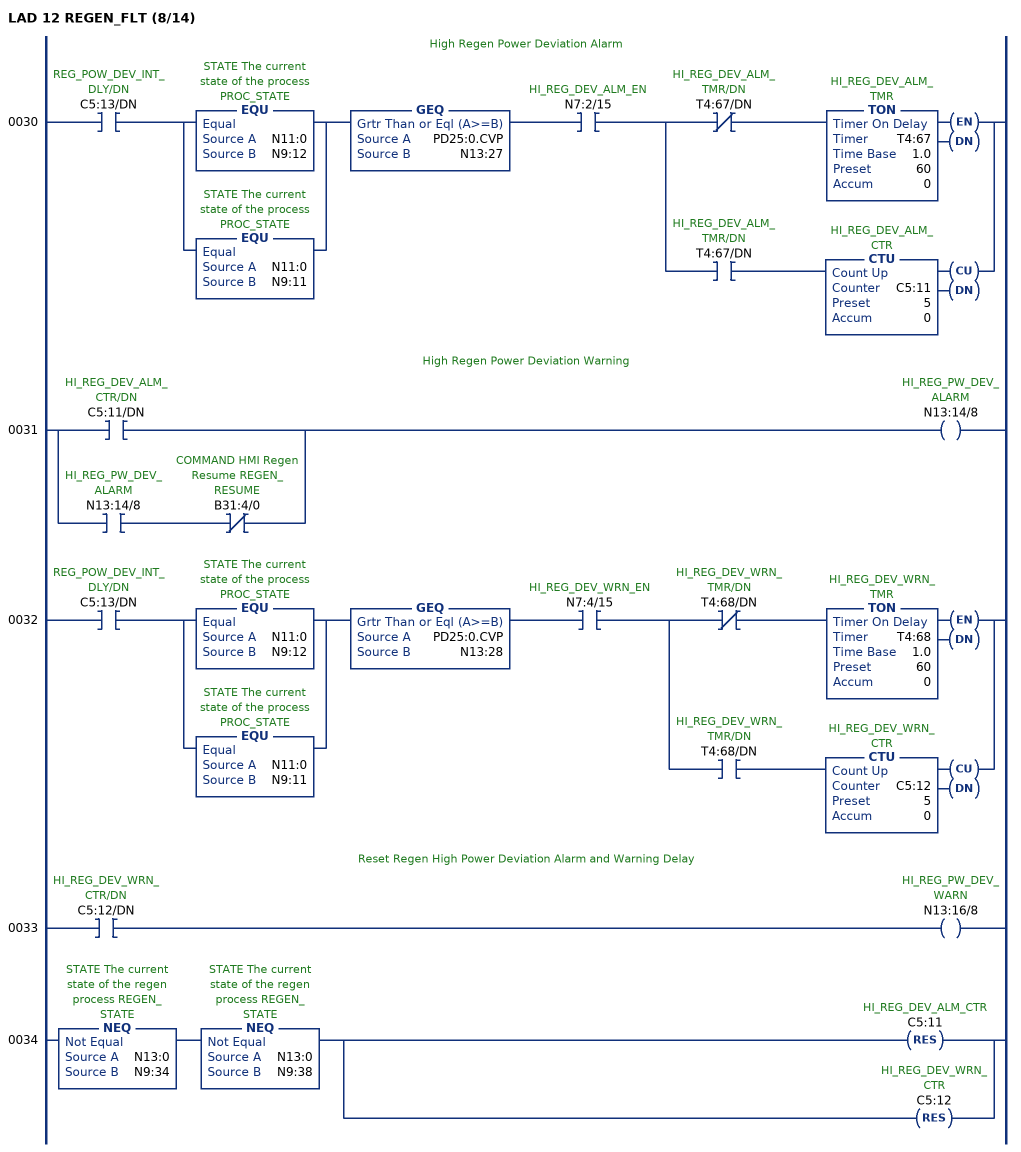
% Rung: 30 %
% High Regen Power Deviation Alarm %
SOR XIC C5:13/DN BST EQU N11:0 N9:12 NXB EQU N11:0 N9:11 BND GEQ PD25:0.CVP N13:27 XIC N7:2/15 BST XIO T4:67/DN TON T4:67 1.0 60 0 NXB XIC T4:67/DN CTU C5:11 5 0 BND EOR
%   C5:13  REG_POW_DEV_INT_DLY %
%   N11:0  PROC_STATE  "STATE The current state of the process" %
%   N9:12  PROC_PURIFY_B  "STATE Process Purify B" %
%   N9:11  PROC_PURIFY_A  "STATE Process Purify A" %
%   N13:27  HI_REG_DEV_ALM_SP %
%   N7:2/15  HI_REG_DEV_ALM_EN %
%   T4:67  HI_REG_DEV_ALM_TMR %
%   C5:11  HI_REG_DEV_ALM_CTR %
% Rung: 31 %
% High Regen Power Deviation Warning %
SOR BST XIC C5:11/DN NXB XIC N13:14/8 XIO B31:4/0 BND OTE N13:14/8 EOR
%   C5:11  HI_REG_DEV_ALM_CTR %
%   N13:14/8  HI_REG_PW_DEV_ALARM %
%   B31:4/0  REGEN_RESUME  "COMMAND HMI Regen Resume" %
% Rung: 32 %
SOR XIC C5:13/DN BST EQU N11:0 N9:12 NXB EQU N11:0 N9:11 BND GEQ PD25:0.CVP N13:28 XIC N7:4/15 BST XIO T4:68/DN TON T4:68 1.0 60 0 NXB XIC T4:68/DN CTU C5:12 5 0 BND EOR
%   C5:13  REG_POW_DEV_INT_DLY %
%   N11:0  PROC_STATE  "STATE The current state of the process" %
%   N9:12  PROC_PURIFY_B  "STATE Process Purify B" %
%   N9:11  PROC_PURIFY_A  "STATE Process Purify A" %
%   N13:28  HI_REG_DEV_WRN_SP %
%   N7:4/15  HI_REG_DEV_WRN_EN %
%   T4:68  HI_REG_DEV_WRN_TMR %
%   C5:12  HI_REG_DEV_WRN_CTR %
% Rung: 33 %
% Reset Regen High Power Deviation Alarm and Warning Delay %
SOR XIC C5:12/DN OTE N13:16/8 EOR
%   C5:12  HI_REG_DEV_WRN_CTR %
%   N13:16/8  HI_REG_PW_DEV_WARN %
% Rung: 34 %
SOR NEQ N13:0 N9:34 NEQ N13:0 N9:38 BST RES C5:11 NXB RES C5:12 BND EOR
%   N13:0  REGEN_STATE  "STATE The current state of the regen process" %
%   N9:34  REGEN_H2_REDUCTION  "STATE Regen Running" %
%   N9:38  REGEN_PURGE  "STATE Regen Hot Purge" %
%   C5:11  HI_REG_DEV_ALM_CTR %
%   C5:12  HI_REG_DEV_WRN_CTR %

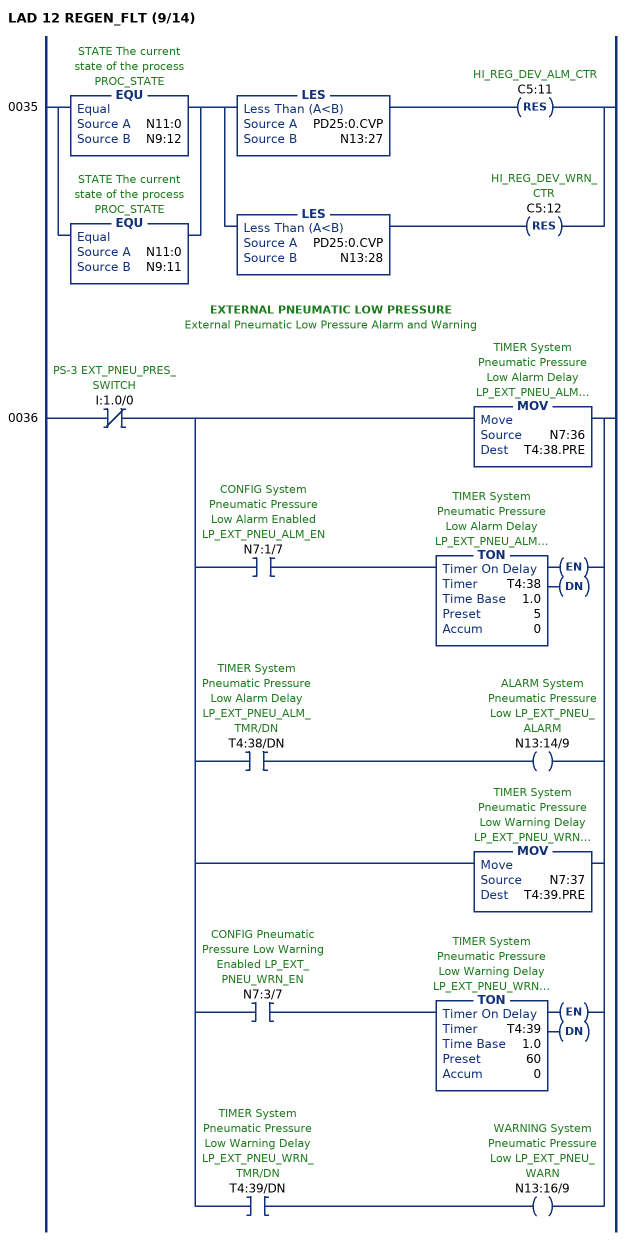
% Rung: 35 %
SOR BST EQU N11:0 N9:12 NXB EQU N11:0 N9:11 BND BST LES PD25:0.CVP N13:27 RES C5:11 NXB LES PD25:0.CVP N13:28 RES C5:12 BND EOR
%   N11:0  PROC_STATE  "STATE The current state of the process" %
%   N9:12  PROC_PURIFY_B  "STATE Process Purify B" %
%   N9:11  PROC_PURIFY_A  "STATE Process Purify A" %
%   N13:27  HI_REG_DEV_ALM_SP %
%   C5:11  HI_REG_DEV_ALM_CTR %
%   N13:28  HI_REG_DEV_WRN_SP %
%   C5:12  HI_REG_DEV_WRN_CTR %
% Rung: 36 %
% TITLE: EXTERNAL PNEUMATIC LOW PRESSURE %
% External Pneumatic Low Pressure Alarm and Warning %
SOR XIO I:1.0/0 BST MOV N7:36 T4:38.PRE NXB XIC N7:1/7 TON T4:38 1.0 5 0 NXB XIC T4:38/DN OTE N13:14/9 NXB MOV N7:37 T4:39.PRE NXB XIC N7:3/7 TON T4:39 1.0 60 0 NXB XIC T4:39/DN OTE N13:16/9 BND EOR
%   I:1.0/0  EXT_PNEU_PRES_SWITCH  "PS-3" %
%   N7:36  LP_EXT_PNEU_ALM_DLY  "CONFIG Pneumatic Pressure Low Alarm Delay" %
%   T4:38  LP_EXT_PNEU_ALM_TMR  "TIMER System Pneumatic Pressure Low Alarm Delay" %
%   N7:1/7  LP_EXT_PNEU_ALM_EN  "CONFIG System Pneumatic Pressure Low Alarm Enabled" %
%   N13:14/9  LP_EXT_PNEU_ALARM  "ALARM System Pneumatic Pressure Low" %
%   N7:37  LP_EXT_PNEU_WRN_DLY  "CONFIG Pneumatic Pressure Low Warning Delay" %
%   T4:39  LP_EXT_PNEU_WRN_TMR  "TIMER System Pneumatic Pressure Low Warning Delay" %
%   N7:3/7  LP_EXT_PNEU_WRN_EN  "CONFIG Pneumatic Pressure Low Warning Enabled" %
%   N13:16/9  LP_EXT_PNEU_WARN  "WARNING System Pneumatic Pressure Low" %

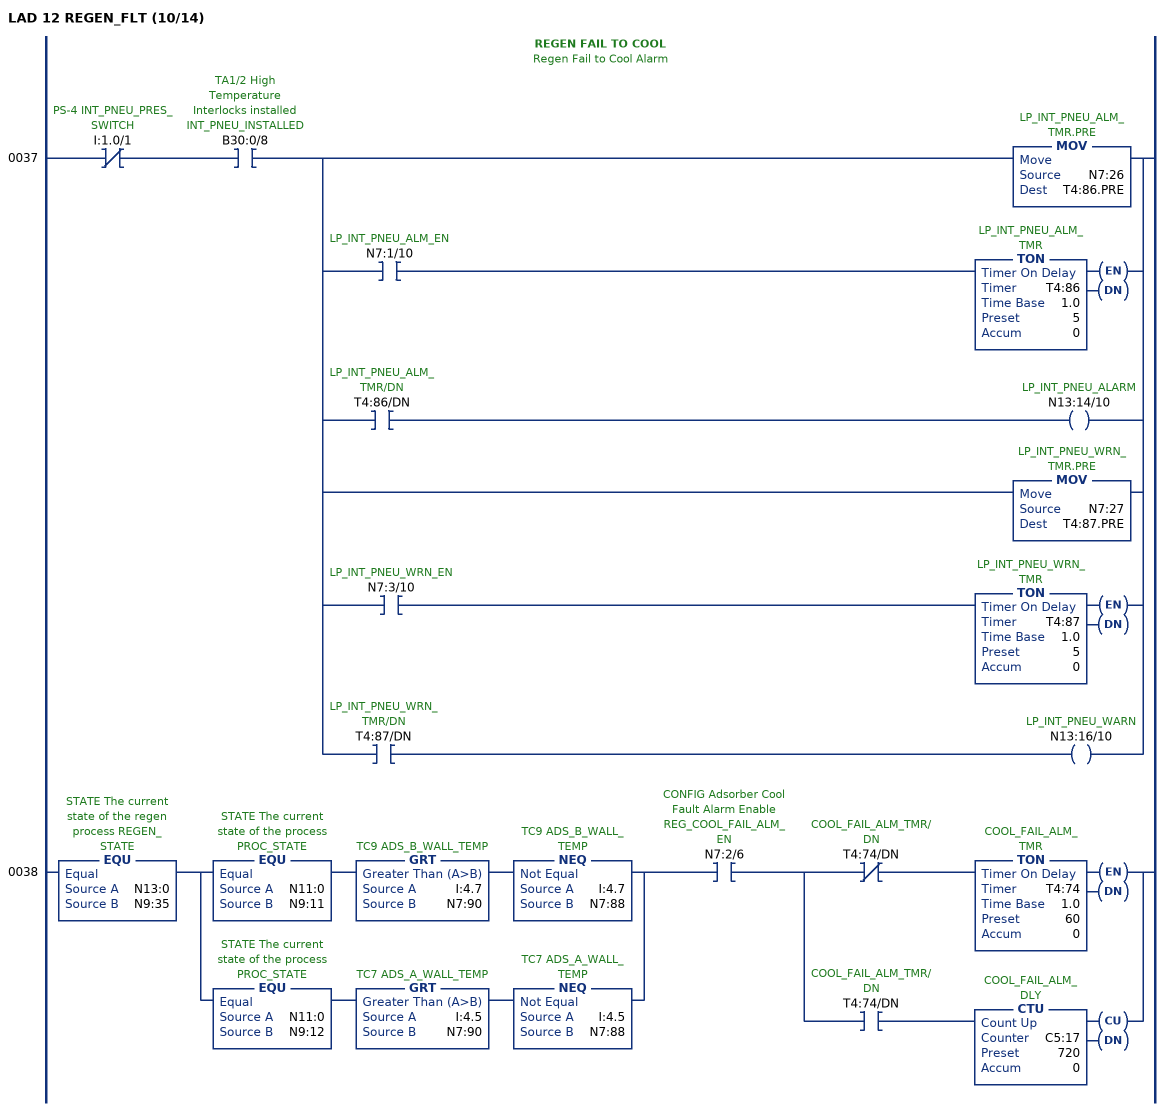
% Rung: 37 %
% TITLE: REGEN FAIL TO COOL %
% Regen Fail to Cool Alarm %
SOR XIO I:1.0/1 XIC B30:0/8 BST MOV N7:26 T4:86.PRE NXB XIC N7:1/10 TON T4:86 1.0 5 0 NXB XIC T4:86/DN OTE N13:14/10 NXB MOV N7:27 T4:87.PRE NXB XIC N7:3/10 TON T4:87 1.0 5 0 NXB XIC T4:87/DN OTE N13:16/10 BND EOR
%   I:1.0/1  INT_PNEU_PRES_SWITCH  "PS-4" %
%   B30:0/8  INT_PNEU_INSTALLED  "TA1/2 High Temperature Interlocks installed" %
%   N7:26  LP_INT_PNEU_ALM_DLY %
%   T4:86  LP_INT_PNEU_ALM_TMR %
%   N7:1/10  LP_INT_PNEU_ALM_EN %
%   N13:14/10  LP_INT_PNEU_ALARM %
%   N7:27  LP_INT_PNEU_WRN_DLY %
%   T4:87  LP_INT_PNEU_WRN_TMR %
%   N7:3/10  LP_INT_PNEU_WRN_EN %
%   N13:16/10  LP_INT_PNEU_WARN %
% Rung: 38 %
SOR EQU N13:0 N9:35 BST EQU N11:0 N9:11 GRT I:4.7 N7:90 NEQ I:4.7 N7:88 NXB EQU N11:0 N9:12 GRT I:4.5 N7:90 NEQ I:4.5 N7:88 BND XIC N7:2/6 BST XIO T4:74/DN TON T4:74 1.0 60 0 NXB XIC T4:74/DN CTU C5:17 720 0 BND EOR
%   N13:0  REGEN_STATE  "STATE The current state of the regen process" %
%   N9:35  REGEN_COOL_WALL  "STATE Regen Cool wall" %
%   N11:0  PROC_STATE  "STATE The current state of the process" %
%   N9:11  PROC_PURIFY_A  "STATE Process Purify A" %
%   I:4.7  ADS_B_WALL_TEMP  "TC9" %
%   N7:90  REG_COOL_FAIL_ALM_SP %
%   N7:88  TC_OPEN_SP  "CONFIG The value read by an open TC input" %
%   N9:12  PROC_PURIFY_B  "STATE Process Purify B" %
%   I:4.5  ADS_A_WALL_TEMP  "TC7" %
%   N7:2/6  REG_COOL_FAIL_ALM_EN  "CONFIG Adsorber Cool Fault Alarm Enable" %
%   T4:74  COOL_FAIL_ALM_TMR %
%   C5:17  COOL_FAIL_ALM_DLY %

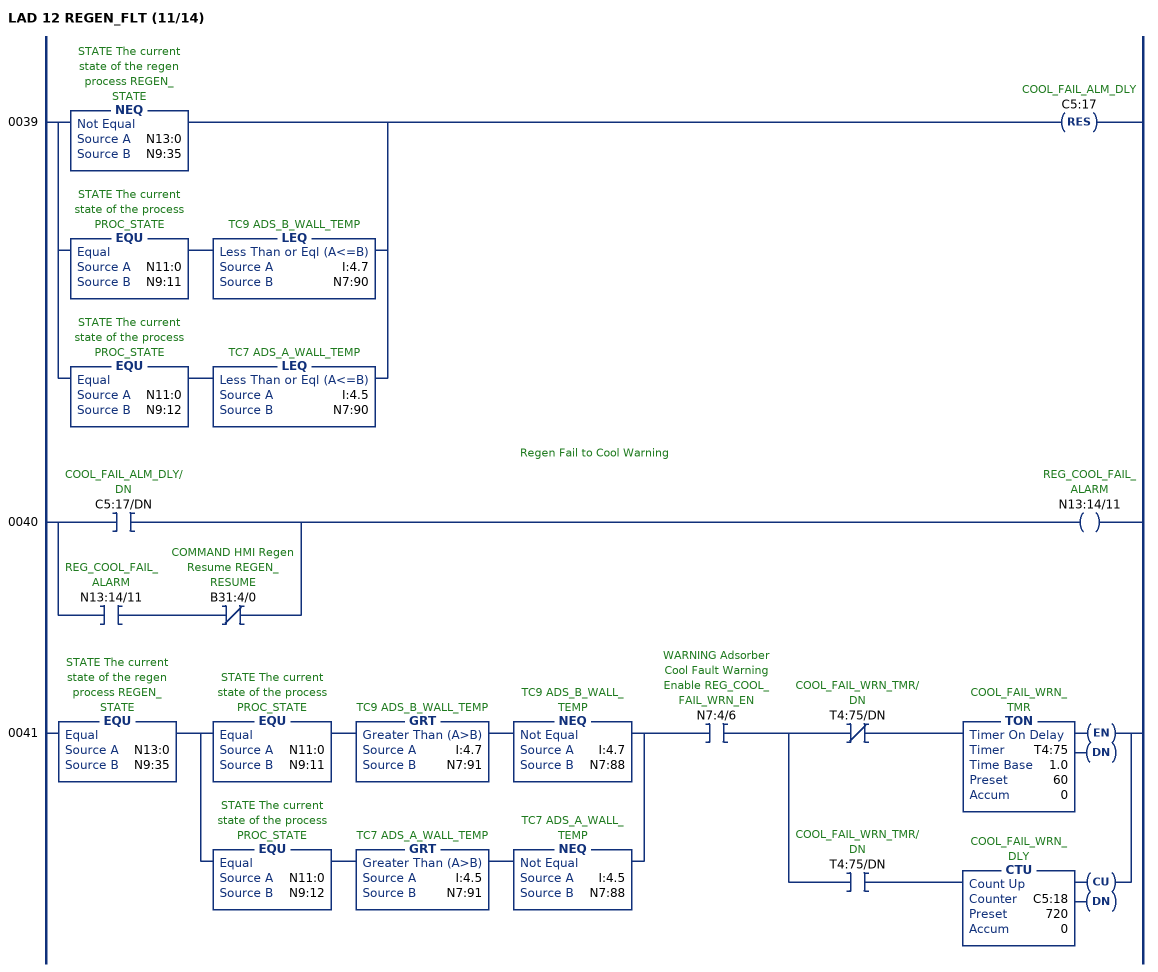
% Rung: 39 %
SOR BST NEQ N13:0 N9:35 NXB EQU N11:0 N9:11 LEQ I:4.7 N7:90 NXB EQU N11:0 N9:12 LEQ I:4.5 N7:90 BND RES C5:17 EOR
%   N13:0  REGEN_STATE  "STATE The current state of the regen process" %
%   N9:35  REGEN_COOL_WALL  "STATE Regen Cool wall" %
%   N11:0  PROC_STATE  "STATE The current state of the process" %
%   N9:11  PROC_PURIFY_A  "STATE Process Purify A" %
%   I:4.7  ADS_B_WALL_TEMP  "TC9" %
%   N7:90  REG_COOL_FAIL_ALM_SP %
%   N9:12  PROC_PURIFY_B  "STATE Process Purify B" %
%   I:4.5  ADS_A_WALL_TEMP  "TC7" %
%   C5:17  COOL_FAIL_ALM_DLY %
% Rung: 40 %
% Regen Fail to Cool Warning %
SOR BST XIC C5:17/DN NXB XIC N13:14/11 XIO B31:4/0 BND OTE N13:14/11 EOR
%   C5:17  COOL_FAIL_ALM_DLY %
%   N13:14/11  REG_COOL_FAIL_ALARM %
%   B31:4/0  REGEN_RESUME  "COMMAND HMI Regen Resume" %
% Rung: 41 %
SOR EQU N13:0 N9:35 BST EQU N11:0 N9:11 GRT I:4.7 N7:91 NEQ I:4.7 N7:88 NXB EQU N11:0 N9:12 GRT I:4.5 N7:91 NEQ I:4.5 N7:88 BND XIC N7:4/6 BST XIO T4:75/DN TON T4:75 1.0 60 0 NXB XIC T4:75/DN CTU C5:18 720 0 BND EOR
%   N13:0  REGEN_STATE  "STATE The current state of the regen process" %
%   N9:35  REGEN_COOL_WALL  "STATE Regen Cool wall" %
%   N11:0  PROC_STATE  "STATE The current state of the process" %
%   N9:11  PROC_PURIFY_A  "STATE Process Purify A" %
%   I:4.7  ADS_B_WALL_TEMP  "TC9" %
%   N7:91  REG_COOL_FAIL_WRN_SP %
%   N7:88  TC_OPEN_SP  "CONFIG The value read by an open TC input" %
%   N9:12  PROC_PURIFY_B  "STATE Process Purify B" %
%   I:4.5  ADS_A_WALL_TEMP  "TC7" %
%   N7:4/6  REG_COOL_FAIL_WRN_EN  "WARNING Adsorber Cool Fault Warning Enable" %
%   T4:75  COOL_FAIL_WRN_TMR %
%   C5:18  COOL_FAIL_WRN_DLY %

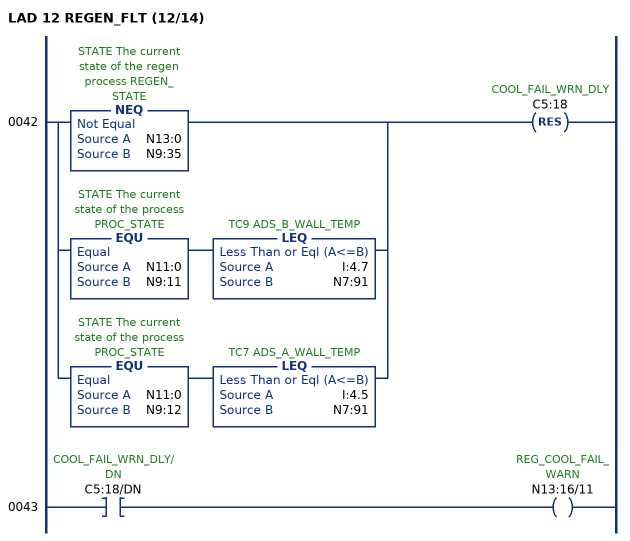
% Rung: 42 %
SOR BST NEQ N13:0 N9:35 NXB EQU N11:0 N9:11 LEQ I:4.7 N7:91 NXB EQU N11:0 N9:12 LEQ I:4.5 N7:91 BND RES C5:18 EOR
%   N13:0  REGEN_STATE  "STATE The current state of the regen process" %
%   N9:35  REGEN_COOL_WALL  "STATE Regen Cool wall" %
%   N11:0  PROC_STATE  "STATE The current state of the process" %
%   N9:11  PROC_PURIFY_A  "STATE Process Purify A" %
%   I:4.7  ADS_B_WALL_TEMP  "TC9" %
%   N7:91  REG_COOL_FAIL_WRN_SP %
%   N9:12  PROC_PURIFY_B  "STATE Process Purify B" %
%   I:4.5  ADS_A_WALL_TEMP  "TC7" %
%   C5:18  COOL_FAIL_WRN_DLY %
% Rung: 43 %
SOR XIC C5:18/DN OTE N13:16/11 EOR
%   C5:18  COOL_FAIL_WRN_DLY %
%   N13:16/11  REG_COOL_FAIL_WARN %

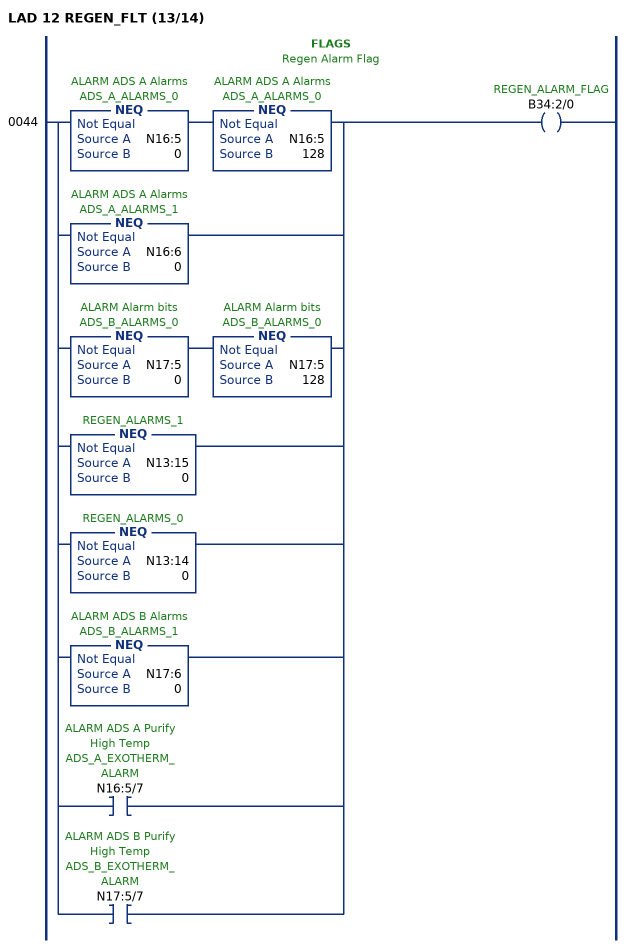
% Rung: 44 %
% TITLE: FLAGS %
% Regen Alarm Flag %
SOR BST NEQ N16:5 0 NEQ N16:5 128 NXB NEQ N16:6 0 NXB NEQ N17:5 0 NEQ N17:5 128 NXB NEQ N13:15 0 NXB NEQ N13:14 0 NXB NEQ N17:6 0 NXB XIC N16:5/7 NXB XIC N17:5/7 BND OTE B34:2/0 EOR
%   N16:5  ADS_A_ALARMS_0  "ALARM ADS A Alarms" %
%   N16:6  ADS_A_ALARMS_1  "ALARM ADS A Alarms" %
%   N17:5  ADS_B_ALARMS_0  "ALARM Alarm bits" %
%   N13:15  REGEN_ALARMS_1 %
%   N13:14  REGEN_ALARMS_0 %
%   N17:6  ADS_B_ALARMS_1  "ALARM ADS B Alarms" %
%   N16:5/7  ADS_A_EXOTHERM_ALARM  "ALARM ADS A Purify High Temp" %
%   N17:5/7  ADS_B_EXOTHERM_ALARM  "ALARM ADS B Purify High Temp" %
%   B34:2/0  REGEN_ALARM_FLAG %

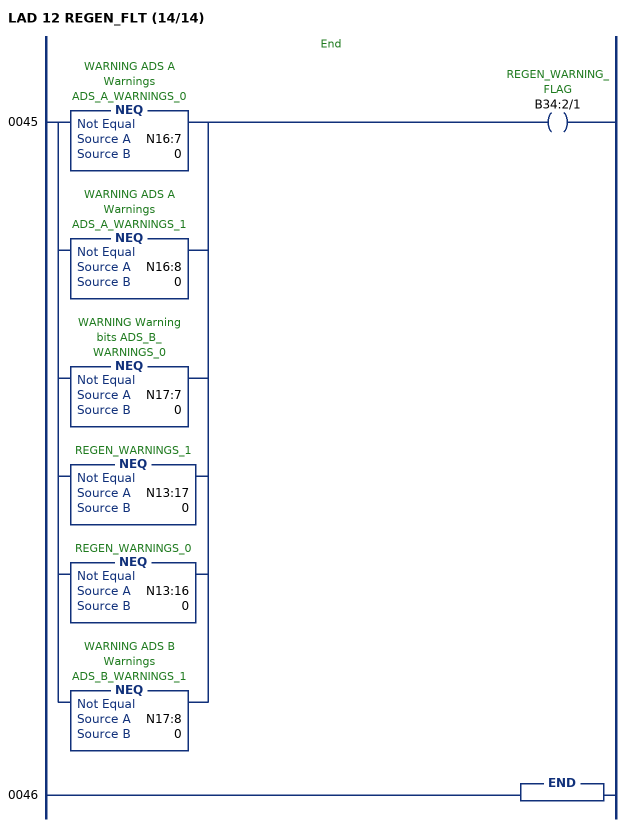
% Rung: 45 %
% End %
SOR BST NEQ N16:7 0 NXB NEQ N16:8 0 NXB NEQ N17:7 0 NXB NEQ N13:17 0 NXB NEQ N13:16 0 NXB NEQ N17:8 0 BND OTE B34:2/1 EOR
%   N16:7  ADS_A_WARNINGS_0  "WARNING ADS A Warnings" %
%   N16:8  ADS_A_WARNINGS_1  "WARNING ADS A Warnings" %
%   N17:7  ADS_B_WARNINGS_0  "WARNING Warning bits" %
%   N13:17  REGEN_WARNINGS_1 %
%   N13:16  REGEN_WARNINGS_0 %
%   N17:8  ADS_B_WARNINGS_1  "WARNING ADS B Warnings" %
%   B34:2/1  REGEN_WARNING_FLAG %
% Rung: 46 %
SOR END EOR

LADDER 17 "BYPASS"    % Controls the bypass %
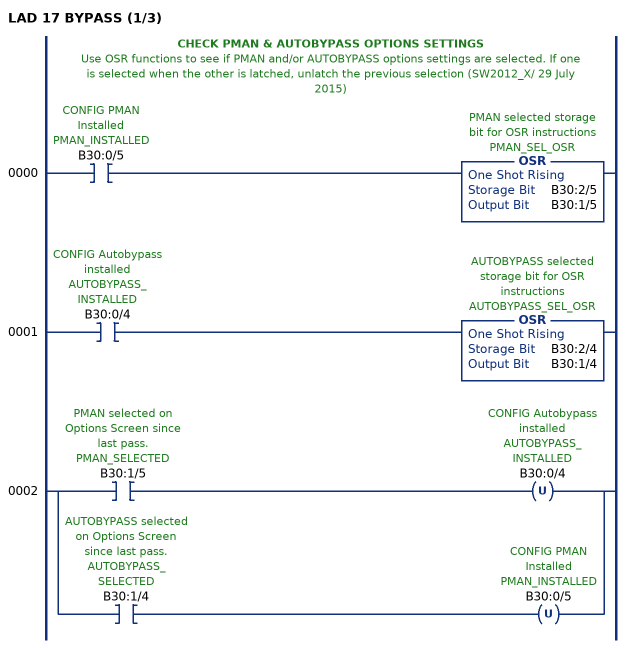
% Rung: 0 %
% TITLE: CHECK PMAN & AUTOBYPASS OPTIONS SETTINGS %
% Use OSR functions to see if PMAN and/or AUTOBYPASS options settings are selected. If one is selected when the other is latched, unlatch the previous selection (SW2012_X/ 29 July 2015) %
SOR XIC B30:0/5 OSR B30:2/5 B30:1/5 EOR
%   B30:0/5  PMAN_INSTALLED  "CONFIG PMAN Installed" %
%   B30:2/5  PMAN_SEL_OSR  "PMAN selected storage bit for OSR instructions" %
%   B30:1/5  PMAN_SELECTED  "PMAN selected on Options Screen since last pass." %
% Rung: 1 %
SOR XIC B30:0/4 OSR B30:2/4 B30:1/4 EOR
%   B30:0/4  AUTOBYPASS_INSTALLED  "CONFIG Autobypass installed" %
%   B30:2/4  AUTOBYPASS_SEL_OSR  "AUTOBYPASS selected storage bit for OSR instructions" %
%   B30:1/4  AUTOBYPASS_SELECTED  "AUTOBYPASS selected on Options Screen since last pass." %
% Rung: 2 %
SOR BST XIC B30:1/5 OTU B30:0/4 NXB XIC B30:1/4 OTU B30:0/5 BND EOR
%   B30:1/5  PMAN_SELECTED  "PMAN selected on Options Screen since last pass." %
%   B30:0/4  AUTOBYPASS_INSTALLED  "CONFIG Autobypass installed" %
%   B30:1/4  AUTOBYPASS_SELECTED  "AUTOBYPASS selected on Options Screen since last pass." %
%   B30:0/5  PMAN_INSTALLED  "CONFIG PMAN Installed" %

